REGION Network 171: CIP Return Pump Using P-08.02 (Speed)
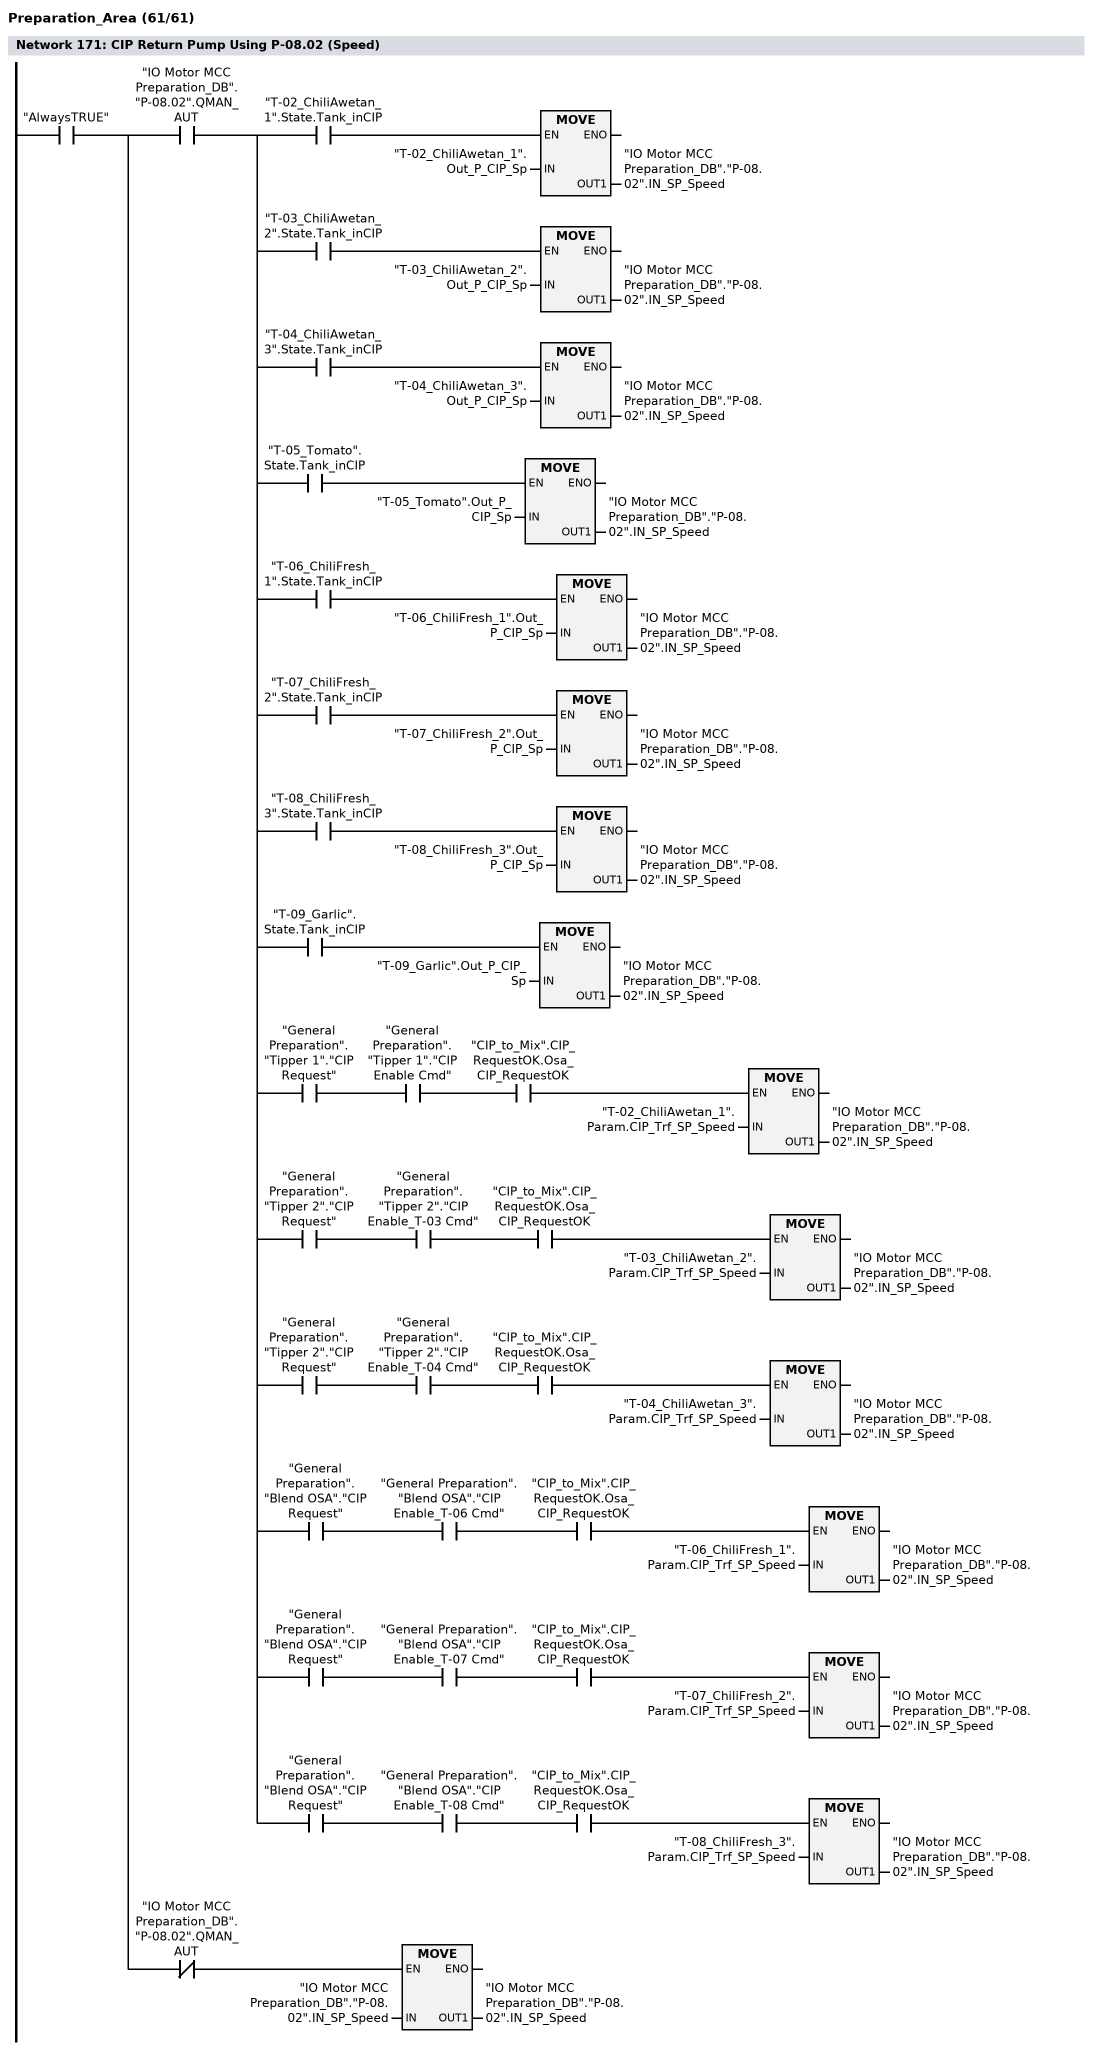
   RUNG wire#powerrail
      Contact( "AlwaysTRUE" )
      wire#w1
      Contact( "IO Motor MCC Preparation_DB"."P-08.02".QMAN_AUT )
      wire#w2
      Contact( "T-02_ChiliAwetan_1".State.Tank_inCIP )
      Move(in := "T-02_ChiliAwetan_1".Out_P_CIP_Sp, out1 => "IO Motor MCC Preparation_DB"."P-08.02".IN_SP_Speed)
   END_RUNG
   RUNG wire#w2
      Contact( "T-03_ChiliAwetan_2".State.Tank_inCIP )
      Move(in := "T-03_ChiliAwetan_2".Out_P_CIP_Sp, out1 => "IO Motor MCC Preparation_DB"."P-08.02".IN_SP_Speed)
   END_RUNG
   RUNG wire#w2
      Contact( "T-04_ChiliAwetan_3".State.Tank_inCIP )
      Move(in := "T-04_ChiliAwetan_3".Out_P_CIP_Sp, out1 => "IO Motor MCC Preparation_DB"."P-08.02".IN_SP_Speed)
   END_RUNG
   RUNG wire#w2
      Contact( "T-05_Tomato".State.Tank_inCIP )
      Move(in := "T-05_Tomato".Out_P_CIP_Sp, out1 => "IO Motor MCC Preparation_DB"."P-08.02".IN_SP_Speed)
   END_RUNG
   RUNG wire#w2
      Contact( "T-06_ChiliFresh_1".State.Tank_inCIP )
      Move(in := "T-06_ChiliFresh_1".Out_P_CIP_Sp, out1 => "IO Motor MCC Preparation_DB"."P-08.02".IN_SP_Speed)
   END_RUNG
   RUNG wire#w2
      Contact( "T-07_ChiliFresh_2".State.Tank_inCIP )
      Move(in := "T-07_ChiliFresh_2".Out_P_CIP_Sp, out1 => "IO Motor MCC Preparation_DB"."P-08.02".IN_SP_Speed)
   END_RUNG
   RUNG wire#w2
      Contact( "T-08_ChiliFresh_3".State.Tank_inCIP )
      Move(in := "T-08_ChiliFresh_3".Out_P_CIP_Sp, out1 => "IO Motor MCC Preparation_DB"."P-08.02".IN_SP_Speed)
   END_RUNG
   RUNG wire#w2
      Contact( "T-09_Garlic".State.Tank_inCIP )
      Move(in := "T-09_Garlic".Out_P_CIP_Sp, out1 => "IO Motor MCC Preparation_DB"."P-08.02".IN_SP_Speed)
   END_RUNG
   RUNG wire#w2
      Contact( "General Preparation"."Tipper 1"."CIP Request" )
      Contact( "General Preparation"."Tipper 1"."CIP Enable Cmd" )
      Contact( "CIP_to_Mix".CIP_RequestOK.Osa_CIP_RequestOK )
      Move(in := "T-02_ChiliAwetan_1".Param.CIP_Trf_SP_Speed, out1 => "IO Motor MCC Preparation_DB"."P-08.02".IN_SP_Speed)
   END_RUNG
   RUNG wire#w2
      Contact( "General Preparation"."Tipper 2"."CIP Request" )
      Contact( "General Preparation"."Tipper 2"."CIP Enable_T-03 Cmd" )
      Contact( "CIP_to_Mix".CIP_RequestOK.Osa_CIP_RequestOK )
      Move(in := "T-03_ChiliAwetan_2".Param.CIP_Trf_SP_Speed, out1 => "IO Motor MCC Preparation_DB"."P-08.02".IN_SP_Speed)
   END_RUNG
   RUNG wire#w2
      Contact( "General Preparation"."Tipper 2"."CIP Request" )
      Contact( "General Preparation"."Tipper 2"."CIP Enable_T-04 Cmd" )
      Contact( "CIP_to_Mix".CIP_RequestOK.Osa_CIP_RequestOK )
      Move(in := "T-04_ChiliAwetan_3".Param.CIP_Trf_SP_Speed, out1 => "IO Motor MCC Preparation_DB"."P-08.02".IN_SP_Speed)
   END_RUNG
   RUNG wire#w2
      Contact( "General Preparation"."Blend OSA"."CIP Request" )
      Contact( "General Preparation"."Blend OSA"."CIP Enable_T-06 Cmd" )
      Contact( "CIP_to_Mix".CIP_RequestOK.Osa_CIP_RequestOK )
      Move(in := "T-06_ChiliFresh_1".Param.CIP_Trf_SP_Speed, out1 => "IO Motor MCC Preparation_DB"."P-08.02".IN_SP_Speed)
   END_RUNG
   RUNG wire#w2
      Contact( "General Preparation"."Blend OSA"."CIP Request" )
      Contact( "General Preparation"."Blend OSA"."CIP Enable_T-07 Cmd" )
      Contact( "CIP_to_Mix".CIP_RequestOK.Osa_CIP_RequestOK )
      Move(in := "T-07_ChiliFresh_2".Param.CIP_Trf_SP_Speed, out1 => "IO Motor MCC Preparation_DB"."P-08.02".IN_SP_Speed)
   END_RUNG
   RUNG wire#w2
      Contact( "General Preparation"."Blend OSA"."CIP Request" )
      Contact( "General Preparation"."Blend OSA"."CIP Enable_T-08 Cmd" )
      Contact( "CIP_to_Mix".CIP_RequestOK.Osa_CIP_RequestOK )
      Move(in := "T-08_ChiliFresh_3".Param.CIP_Trf_SP_Speed, out1 => "IO Motor MCC Preparation_DB"."P-08.02".IN_SP_Speed)
   END_RUNG
   RUNG wire#w1
      I_Contact( "IO Motor MCC Preparation_DB"."P-08.02".QMAN_AUT )
      Move(in := "IO Motor MCC Preparation_DB"."P-08.02".IN_SP_Speed, out1 => "IO Motor MCC Preparation_DB"."P-08.02".IN_SP_Speed)
   END_RUNG
   // the same network as SCL:
   #_w1 := "AlwaysTRUE" AND "IO Motor MCC Preparation_DB"."P-08.02".QMAN_AUT;
   IF #_w1 AND "T-02_ChiliAwetan_1".State.Tank_inCIP THEN
       "IO Motor MCC Preparation_DB"."P-08.02".IN_SP_Speed := "T-02_ChiliAwetan_1".Out_P_CIP_Sp;
   END_IF;
   IF #_w1 AND "T-03_ChiliAwetan_2".State.Tank_inCIP THEN
       "IO Motor MCC Preparation_DB"."P-08.02".IN_SP_Speed := "T-03_ChiliAwetan_2".Out_P_CIP_Sp;
   END_IF;
   IF #_w1 AND "T-04_ChiliAwetan_3".State.Tank_inCIP THEN
       "IO Motor MCC Preparation_DB"."P-08.02".IN_SP_Speed := "T-04_ChiliAwetan_3".Out_P_CIP_Sp;
   END_IF;
   IF #_w1 AND "T-05_Tomato".State.Tank_inCIP THEN
       "IO Motor MCC Preparation_DB"."P-08.02".IN_SP_Speed := "T-05_Tomato".Out_P_CIP_Sp;
   END_IF;
   IF #_w1 AND "T-06_ChiliFresh_1".State.Tank_inCIP THEN
       "IO Motor MCC Preparation_DB"."P-08.02".IN_SP_Speed := "T-06_ChiliFresh_1".Out_P_CIP_Sp;
   END_IF;
   IF #_w1 AND "T-07_ChiliFresh_2".State.Tank_inCIP THEN
       "IO Motor MCC Preparation_DB"."P-08.02".IN_SP_Speed := "T-07_ChiliFresh_2".Out_P_CIP_Sp;
   END_IF;
   IF #_w1 AND "T-08_ChiliFresh_3".State.Tank_inCIP THEN
       "IO Motor MCC Preparation_DB"."P-08.02".IN_SP_Speed := "T-08_ChiliFresh_3".Out_P_CIP_Sp;
   END_IF;
   IF #_w1 AND "T-09_Garlic".State.Tank_inCIP THEN
       "IO Motor MCC Preparation_DB"."P-08.02".IN_SP_Speed := "T-09_Garlic".Out_P_CIP_Sp;
   END_IF;
   IF #_w1 AND "General Preparation"."Tipper 1"."CIP Request" AND "General Preparation"."Tipper 1"."CIP Enable Cmd" AND "CIP_to_Mix".CIP_RequestOK.Osa_CIP_RequestOK THEN
       "IO Motor MCC Preparation_DB"."P-08.02".IN_SP_Speed := "T-02_ChiliAwetan_1".Param.CIP_Trf_SP_Speed;
   END_IF;
   IF #_w1 AND "General Preparation"."Tipper 2"."CIP Request" AND "General Preparation"."Tipper 2"."CIP Enable_T-03 Cmd" AND "CIP_to_Mix".CIP_RequestOK.Osa_CIP_RequestOK THEN
       "IO Motor MCC Preparation_DB"."P-08.02".IN_SP_Speed := "T-03_ChiliAwetan_2".Param.CIP_Trf_SP_Speed;
   END_IF;
   IF #_w1 AND "General Preparation"."Tipper 2"."CIP Request" AND "General Preparation"."Tipper 2"."CIP Enable_T-04 Cmd" AND "CIP_to_Mix".CIP_RequestOK.Osa_CIP_RequestOK THEN
       "IO Motor MCC Preparation_DB"."P-08.02".IN_SP_Speed := "T-04_ChiliAwetan_3".Param.CIP_Trf_SP_Speed;
   END_IF;
   IF #_w1 AND "General Preparation"."Blend OSA"."CIP Request" AND "General Preparation"."Blend OSA"."CIP Enable_T-06 Cmd" AND "CIP_to_Mix".CIP_RequestOK.Osa_CIP_RequestOK THEN
       "IO Motor MCC Preparation_DB"."P-08.02".IN_SP_Speed := "T-06_ChiliFresh_1".Param.CIP_Trf_SP_Speed;
   END_IF;
   IF #_w1 AND "General Preparation"."Blend OSA"."CIP Request" AND "General Preparation"."Blend OSA"."CIP Enable_T-07 Cmd" AND "CIP_to_Mix".CIP_RequestOK.Osa_CIP_RequestOK THEN
       "IO Motor MCC Preparation_DB"."P-08.02".IN_SP_Speed := "T-07_ChiliFresh_2".Param.CIP_Trf_SP_Speed;
   END_IF;
   IF #_w1 AND "General Preparation"."Blend OSA"."CIP Request" AND "General Preparation"."Blend OSA"."CIP Enable_T-08 Cmd" AND "CIP_to_Mix".CIP_RequestOK.Osa_CIP_RequestOK THEN
       "IO Motor MCC Preparation_DB"."P-08.02".IN_SP_Speed := "T-08_ChiliFresh_3".Param.CIP_Trf_SP_Speed;
   END_IF;
   IF "AlwaysTRUE" AND NOT "IO Motor MCC Preparation_DB"."P-08.02".QMAN_AUT THEN
       "IO Motor MCC Preparation_DB"."P-08.02".IN_SP_Speed := "IO Motor MCC Preparation_DB"."P-08.02".IN_SP_Speed;
   END_IF;
END_REGION

NETWORK
TITLE = Valve IO
//Valve T-02.01 Chili Awetan Tank 1
      CALL  "IO Valve T02 Chili", "IO_Valve_T02_Chili"
      ( lock    := ,
        Init    := "General_DB".Initial,
        testing := "General_DB"."Testing FB Valve".Preparation,
        Reset   := "General_DB".Reset
      );
//Valve T-03.01 Chili Awetan Tank 2
      CALL  "IO Valve T03 Chili", "IO_Valve_T03_Chili"
      ( lock    := ,
        Init    := "General_DB".Initial,
        testing := "General_DB"."Testing FB Valve".Preparation,
        Reset   := "General_DB".Reset
      );
//Valve T-04.01 Chili Awetan Tank 3
      CALL  "IO Valve T04 Chili", "IO_Valve_T04_Chili"
      ( lock    := ,
        Init    := "General_DB".Initial,
        testing := "General_DB"."Testing FB Valve".Preparation,
        Reset   := "General_DB".Reset
      );
//Valve T-05.01 Tomato Tank
      CALL  "IO Valve T05 Tomato", "IO_Valve_T05_Tomato"
      ( lock    := ,
        Init    := "General_DB".Initial,
        testing := "General_DB"."Testing FB Valve".Preparation,
        Reset   := "General_DB".Reset
      );
//Valve T-06.01 Fresh Chili Tank 1
      CALL  "IO Valve T06 FreshChili", "IO_Valve_T06_FreshChili"
      ( lock    := ,
        Init    := "General_DB".Initial,
        testing := "General_DB"."Testing FB Valve".Preparation,
        Reset   := "General_DB".Reset
      );
//Valve T-07.01 Fresh Chili Tank 2
      CALL  "IO Valve T07 FreshChili", "IO_Valve_T07_FreshChili"
      ( lock    := ,
        Init    := "General_DB".Initial,
        testing := "General_DB"."Testing FB Valve".Preparation,
        Reset   := "General_DB".Reset
      );
//Valve T-08.01 Fresh Chili Tank 3
      CALL  "IO Valve T08 FreshChili", "IO_Valve_T08_FreshChili"
      ( lock    := ,
        Init    := "General_DB".Initial,
        testing := "General_DB"."Testing FB Valve".Preparation,
        Reset   := "General_DB".Reset
      );
//Valve T-09.01 Garlic Tank
      CALL  "IO Valve T09 Garlic", "IO_Valve_T09_Garlic"
      ( lock    := ,
        Init    := "General_DB".Initial,
        testing := "General_DB"."Testing FB Valve".Preparation,
        Reset   := "General_DB".Reset
      );
//Valve T-10.01 Vinegar Tank
      CALL  "IO Valve T10 Vinegar", "IO_Valve_T10_Vinegar"
      ( lock    := ,
        Init    := "General_DB".Initial,
        testing := "General_DB"."Testing FB Valve".Preparation,
        Reset   := "General_DB".Reset
      );
//Valve T-10.01 HotWater
      CALL  "IO Valve T51 HotWaterLine", "IO_Valve_T51_HW"
      ( lock    := ,
        Init    := "General_DB".Initial,
        testing := "General_DB"."Testing FB Valve".Preparation,
        Reset   := "General_DB".Reset
      );


END_FUNCTION

FUNCTION_BLOCK "IO Analog Preparation"   // FB12, LAD
{ S7_Optimized_Access := 'FALSE' }
VERSION : 0.1
// stored: AutoNumber true, IsIECCheckEnabled false, SetENOAutomatically false, UDAEnableTagReadback false
   VAR_INPUT
      Init : Bool;
      Reset : Bool;
   END_VAR
   VAR
      "LT-01.01" : "Ana_w_K1K2";   // LEVEL TRANSMITTER HOT WATER TANK T-01.00
      "TT-01.01" : "Ana_w_K1K2";   // TEMP. TRANSMITTER HOT WATER TANK T-01.00
      "TT-01.02" : "Ana_w_K1K2";   // TEMP.TRANSMITTER LINE HOT WATER
      "LT-02.01" : "Ana_w_K1K2";   // LEVEL TRANSMITTER BUFFER TANK CHILI AWETAN T-02.00
      "LT-03.01" : "Ana_w_K1K2";   // LEVEL TRANSMITTER BUFFER TANK CHILI AWETAN T-03.00
      "LT-04.01" : "Ana_w_K1K2";   // LEVEL TRANSMITTER BUFFER TANK CHILI AWETAN T-04.00
      "LT-05.01" : "Ana_w_K1K2";   // LEVEL TRANSMITTER BUFFER TANK TOMATO T-05.00
      "LT-06.01" : "Ana_w_K1K2";   // LEVEL TRANSMITTER BUFFER TANK CHILI FRESH T-06.00
      "LT-07.01" : "Ana_w_K1K2";   // LEVEL TRANSMITTER BUFFER TANK CHILI FRESH T-07.00
      "LT-08.01" : "Ana_w_K1K2";   // LEVEL TRANSMITTER BUFFER TANK CHILI FRESH T-08.00
      "LT-09.01" : "Ana_w_K1K2";   // LEVEL TRANSMITTER BUFFER TANK GARLIC T-09.00
      "LT-10.01" : "Ana_w_K1K2";   // LEVEL TRANSMITTER BUFFER TANK GARLIC T-10.00
      "TT-51.01" { S7_SetPoint := 'True'} : "Ana_w_K1K2";
      "CV-51.11" { S7_SetPoint := 'True'} : "Ana_w_K1K2";
      "FT-51.01" { S7_SetPoint := 'True'} : "Ana_w_K1K2";
      "FT-02.01" { S7_SetPoint := 'True'} : "Ana_w_K1K2";
      "FT-02.01Com" { S7_SetPoint := 'True'} : "Read FT Comm";
      "FT-03.01" { S7_SetPoint := 'True'} : "Ana_w_K1K2";
      "FT-03.01Com" { S7_SetPoint := 'True'} : "Read FT Comm";
      "FT-04.01" { S7_SetPoint := 'True'} : "Ana_w_K1K2";
      "FT-04.01Com" { S7_SetPoint := 'True'} : "Read FT Comm";
      "FT-05.01" { S7_SetPoint := 'True'} : "Ana_w_K1K2";
      "FT-05.01Com" { S7_SetPoint := 'True'} : "Read FT Comm";
      "FT-06.01" { S7_SetPoint := 'True'} : "Ana_w_K1K2";
      "FT-06.01Com" { S7_SetPoint := 'True'} : "Read FT Comm";
      "FT-07.01" { S7_SetPoint := 'True'} : "Ana_w_K1K2";
      "FT-07.01Com" { S7_SetPoint := 'True'} : "Read FT Comm";
      "FT-08.01" { S7_SetPoint := 'True'} : "Ana_w_K1K2";
      "FT-08.01Com" { S7_SetPoint := 'True'} : "Read FT Comm";
      "FT-09.01" { S7_SetPoint := 'True'} : "Ana_w_K1K2";
      "FT-09.01Com" { S7_SetPoint := 'True'} : "Read FT Comm";
      "FT-10.01" { S7_SetPoint := 'True'} : "Ana_w_K1K2";
      "FT-10.01Com" { S7_SetPoint := 'True'} : "Read FT Comm";
   END_VAR
BEGIN

REGION Network 1: LT-01.01
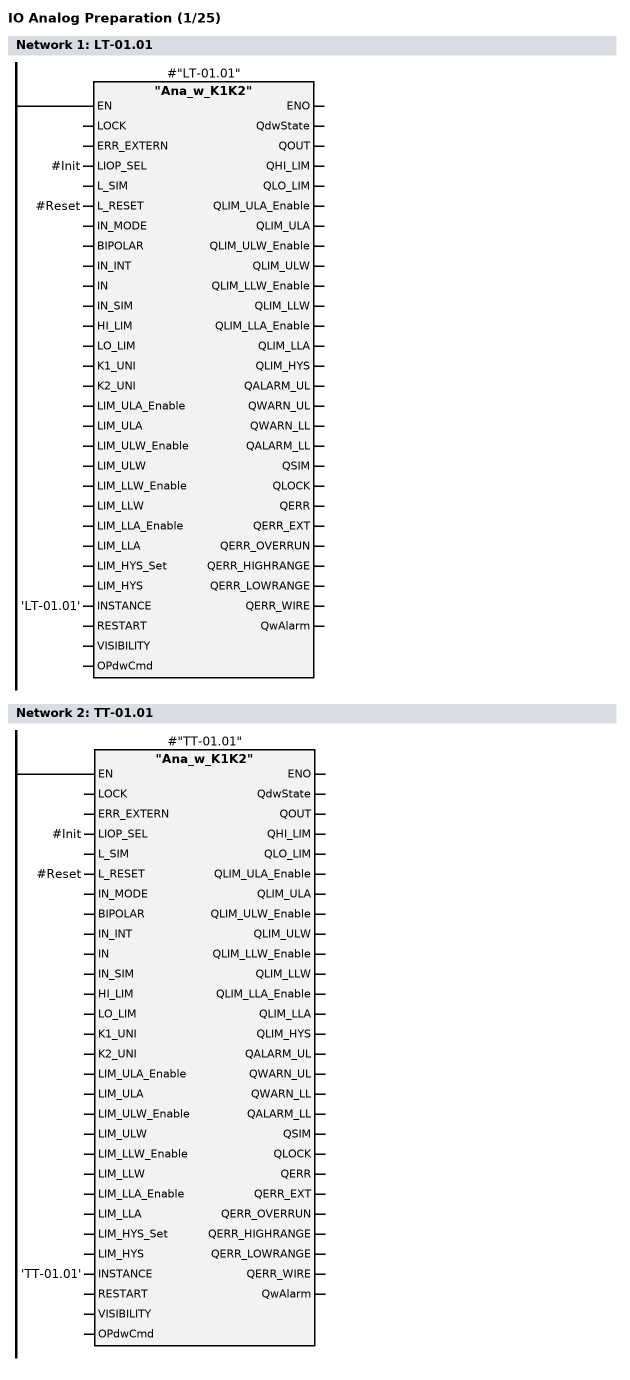
   RUNG wire#powerrail
      #"LT-01.01"(LOCK :=, ERR_EXTERN :=, LIOP_SEL := #Init, L_SIM :=, L_RESET := #Reset, IN_MODE :=, BIPOLAR :=, IN_INT :=, IN :=, IN_SIM :=, HI_LIM :=, LO_LIM :=, K1_UNI :=, K2_UNI :=, LIM_ULA_Enable :=, LIM_ULA :=, LIM_ULW_Enable :=, LIM_ULW :=, LIM_LLW_Enable :=, LIM_LLW :=, LIM_LLA_Enable :=, LIM_LLA :=, LIM_HYS_Set :=, LIM_HYS :=, INSTANCE := 'LT-01.01', RESTART :=, VISIBILITY :=, OPdwCmd :=, QdwState =>, QOUT =>, QHI_LIM =>, QLO_LIM =>, QLIM_ULA_Enable =>, QLIM_ULA =>, QLIM_ULW_Enable =>, QLIM_ULW =>, QLIM_LLW_Enable =>, QLIM_LLW =>, QLIM_LLA_Enable =>, QLIM_LLA =>, QLIM_HYS =>, QALARM_UL =>, QWARN_UL =>, QWARN_LL =>, QALARM_LL =>, QSIM =>, QLOCK =>, QERR =>, QERR_EXT =>, QERR_OVERRUN =>, QERR_HIGHRANGE =>, QERR_LOWRANGE =>, QERR_WIRE =>, QwAlarm =>)
   END_RUNG
   // the same network as SCL:
   #"LT-01.01"(LIOP_SEL := #Init, L_RESET := #Reset, INSTANCE := 'LT-01.01');   // "Ana_w_K1K2"
END_REGION

REGION Network 2: TT-01.01
   RUNG wire#powerrail
      #"TT-01.01"(LOCK :=, ERR_EXTERN :=, LIOP_SEL := #Init, L_SIM :=, L_RESET := #Reset, IN_MODE :=, BIPOLAR :=, IN_INT :=, IN :=, IN_SIM :=, HI_LIM :=, LO_LIM :=, K1_UNI :=, K2_UNI :=, LIM_ULA_Enable :=, LIM_ULA :=, LIM_ULW_Enable :=, LIM_ULW :=, LIM_LLW_Enable :=, LIM_LLW :=, LIM_LLA_Enable :=, LIM_LLA :=, LIM_HYS_Set :=, LIM_HYS :=, INSTANCE := 'TT-01.01', RESTART :=, VISIBILITY :=, OPdwCmd :=, QdwState =>, QOUT =>, QHI_LIM =>, QLO_LIM =>, QLIM_ULA_Enable =>, QLIM_ULA =>, QLIM_ULW_Enable =>, QLIM_ULW =>, QLIM_LLW_Enable =>, QLIM_LLW =>, QLIM_LLA_Enable =>, QLIM_LLA =>, QLIM_HYS =>, QALARM_UL =>, QWARN_UL =>, QWARN_LL =>, QALARM_LL =>, QSIM =>, QLOCK =>, QERR =>, QERR_EXT =>, QERR_OVERRUN =>, QERR_HIGHRANGE =>, QERR_LOWRANGE =>, QERR_WIRE =>, QwAlarm =>)
   END_RUNG
   // the same network as SCL:
   #"TT-01.01"(LIOP_SEL := #Init, L_RESET := #Reset, INSTANCE := 'TT-01.01');   // "Ana_w_K1K2"
END_REGION

REGION Network 3: TT-01.02
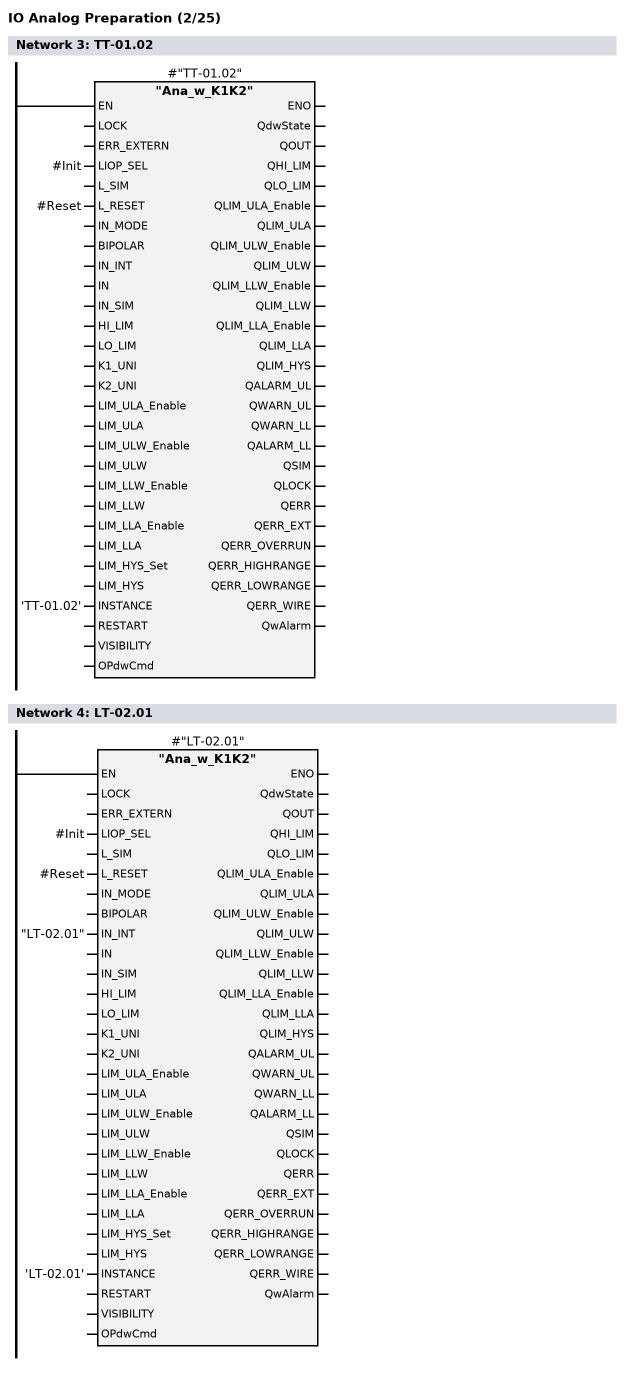
   RUNG wire#powerrail
      #"TT-01.02"(LOCK :=, ERR_EXTERN :=, LIOP_SEL := #Init, L_SIM :=, L_RESET := #Reset, IN_MODE :=, BIPOLAR :=, IN_INT :=, IN :=, IN_SIM :=, HI_LIM :=, LO_LIM :=, K1_UNI :=, K2_UNI :=, LIM_ULA_Enable :=, LIM_ULA :=, LIM_ULW_Enable :=, LIM_ULW :=, LIM_LLW_Enable :=, LIM_LLW :=, LIM_LLA_Enable :=, LIM_LLA :=, LIM_HYS_Set :=, LIM_HYS :=, INSTANCE := 'TT-01.02', RESTART :=, VISIBILITY :=, OPdwCmd :=, QdwState =>, QOUT =>, QHI_LIM =>, QLO_LIM =>, QLIM_ULA_Enable =>, QLIM_ULA =>, QLIM_ULW_Enable =>, QLIM_ULW =>, QLIM_LLW_Enable =>, QLIM_LLW =>, QLIM_LLA_Enable =>, QLIM_LLA =>, QLIM_HYS =>, QALARM_UL =>, QWARN_UL =>, QWARN_LL =>, QALARM_LL =>, QSIM =>, QLOCK =>, QERR =>, QERR_EXT =>, QERR_OVERRUN =>, QERR_HIGHRANGE =>, QERR_LOWRANGE =>, QERR_WIRE =>, QwAlarm =>)
   END_RUNG
   // the same network as SCL:
   #"TT-01.02"(LIOP_SEL := #Init, L_RESET := #Reset, INSTANCE := 'TT-01.02');   // "Ana_w_K1K2"
END_REGION

REGION Network 4: LT-02.01
   RUNG wire#powerrail
      #"LT-02.01"(LOCK :=, ERR_EXTERN :=, LIOP_SEL := #Init, L_SIM :=, L_RESET := #Reset, IN_MODE :=, BIPOLAR :=, IN_INT := "LT-02.01", IN :=, IN_SIM :=, HI_LIM :=, LO_LIM :=, K1_UNI :=, K2_UNI :=, LIM_ULA_Enable :=, LIM_ULA :=, LIM_ULW_Enable :=, LIM_ULW :=, LIM_LLW_Enable :=, LIM_LLW :=, LIM_LLA_Enable :=, LIM_LLA :=, LIM_HYS_Set :=, LIM_HYS :=, INSTANCE := 'LT-02.01', RESTART :=, VISIBILITY :=, OPdwCmd :=, QdwState =>, QOUT =>, QHI_LIM =>, QLO_LIM =>, QLIM_ULA_Enable =>, QLIM_ULA =>, QLIM_ULW_Enable =>, QLIM_ULW =>, QLIM_LLW_Enable =>, QLIM_LLW =>, QLIM_LLA_Enable =>, QLIM_LLA =>, QLIM_HYS =>, QALARM_UL =>, QWARN_UL =>, QWARN_LL =>, QALARM_LL =>, QSIM =>, QLOCK =>, QERR =>, QERR_EXT =>, QERR_OVERRUN =>, QERR_HIGHRANGE =>, QERR_LOWRANGE =>, QERR_WIRE =>, QwAlarm =>)
   END_RUNG
   // the same network as SCL:
   #"LT-02.01"(LIOP_SEL := #Init, L_RESET := #Reset, IN_INT := "LT-02.01", INSTANCE := 'LT-02.01');   // "Ana_w_K1K2"
END_REGION

REGION Network 5: LT-03.01
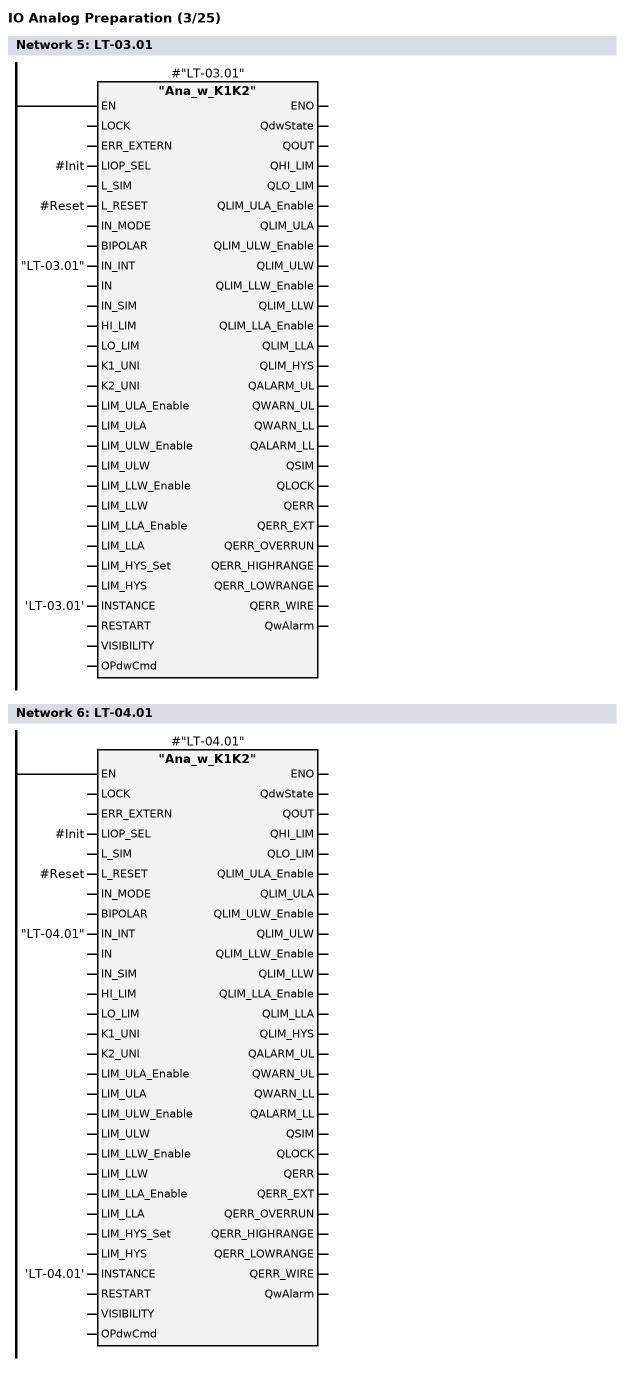
   RUNG wire#powerrail
      #"LT-03.01"(LOCK :=, ERR_EXTERN :=, LIOP_SEL := #Init, L_SIM :=, L_RESET := #Reset, IN_MODE :=, BIPOLAR :=, IN_INT := "LT-03.01", IN :=, IN_SIM :=, HI_LIM :=, LO_LIM :=, K1_UNI :=, K2_UNI :=, LIM_ULA_Enable :=, LIM_ULA :=, LIM_ULW_Enable :=, LIM_ULW :=, LIM_LLW_Enable :=, LIM_LLW :=, LIM_LLA_Enable :=, LIM_LLA :=, LIM_HYS_Set :=, LIM_HYS :=, INSTANCE := 'LT-03.01', RESTART :=, VISIBILITY :=, OPdwCmd :=, QdwState =>, QOUT =>, QHI_LIM =>, QLO_LIM =>, QLIM_ULA_Enable =>, QLIM_ULA =>, QLIM_ULW_Enable =>, QLIM_ULW =>, QLIM_LLW_Enable =>, QLIM_LLW =>, QLIM_LLA_Enable =>, QLIM_LLA =>, QLIM_HYS =>, QALARM_UL =>, QWARN_UL =>, QWARN_LL =>, QALARM_LL =>, QSIM =>, QLOCK =>, QERR =>, QERR_EXT =>, QERR_OVERRUN =>, QERR_HIGHRANGE =>, QERR_LOWRANGE =>, QERR_WIRE =>, QwAlarm =>)
   END_RUNG
   // the same network as SCL:
   #"LT-03.01"(LIOP_SEL := #Init, L_RESET := #Reset, IN_INT := "LT-03.01", INSTANCE := 'LT-03.01');   // "Ana_w_K1K2"
END_REGION

REGION Network 6: LT-04.01
   RUNG wire#powerrail
      #"LT-04.01"(LOCK :=, ERR_EXTERN :=, LIOP_SEL := #Init, L_SIM :=, L_RESET := #Reset, IN_MODE :=, BIPOLAR :=, IN_INT := "LT-04.01", IN :=, IN_SIM :=, HI_LIM :=, LO_LIM :=, K1_UNI :=, K2_UNI :=, LIM_ULA_Enable :=, LIM_ULA :=, LIM_ULW_Enable :=, LIM_ULW :=, LIM_LLW_Enable :=, LIM_LLW :=, LIM_LLA_Enable :=, LIM_LLA :=, LIM_HYS_Set :=, LIM_HYS :=, INSTANCE := 'LT-04.01', RESTART :=, VISIBILITY :=, OPdwCmd :=, QdwState =>, QOUT =>, QHI_LIM =>, QLO_LIM =>, QLIM_ULA_Enable =>, QLIM_ULA =>, QLIM_ULW_Enable =>, QLIM_ULW =>, QLIM_LLW_Enable =>, QLIM_LLW =>, QLIM_LLA_Enable =>, QLIM_LLA =>, QLIM_HYS =>, QALARM_UL =>, QWARN_UL =>, QWARN_LL =>, QALARM_LL =>, QSIM =>, QLOCK =>, QERR =>, QERR_EXT =>, QERR_OVERRUN =>, QERR_HIGHRANGE =>, QERR_LOWRANGE =>, QERR_WIRE =>, QwAlarm =>)
   END_RUNG
   // the same network as SCL:
   #"LT-04.01"(LIOP_SEL := #Init, L_RESET := #Reset, IN_INT := "LT-04.01", INSTANCE := 'LT-04.01');   // "Ana_w_K1K2"
END_REGION

REGION Network 7: LT-05.01
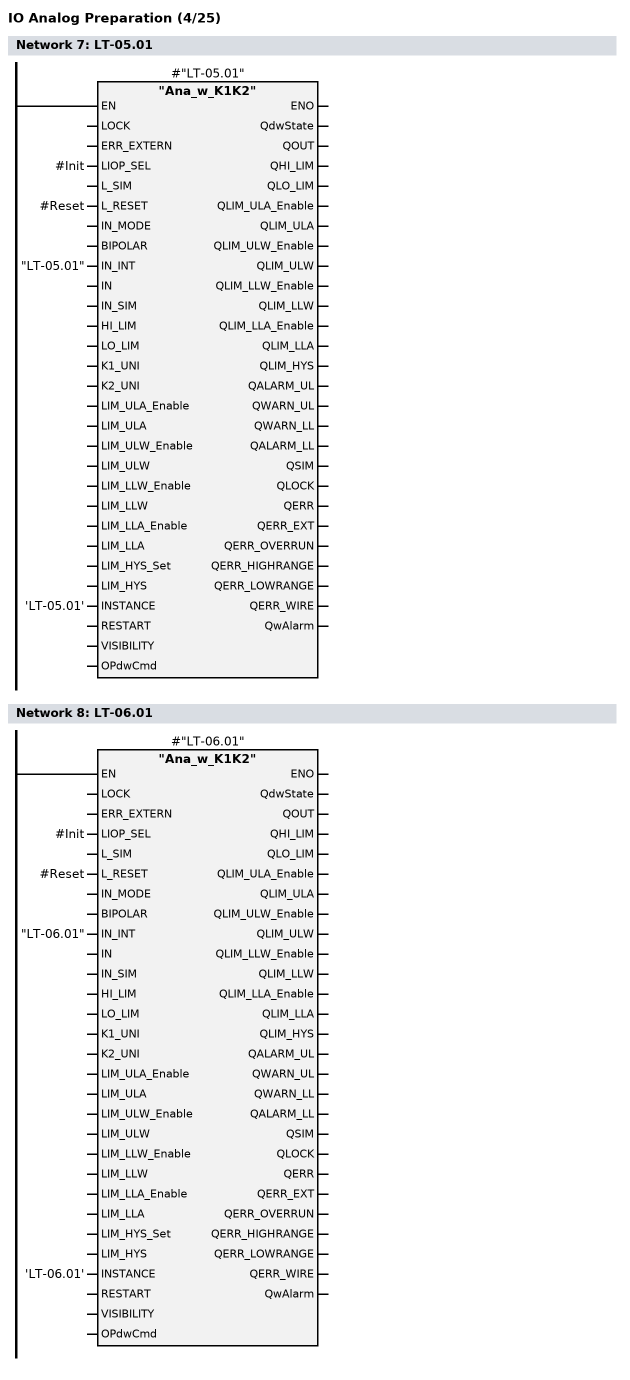
   RUNG wire#powerrail
      #"LT-05.01"(LOCK :=, ERR_EXTERN :=, LIOP_SEL := #Init, L_SIM :=, L_RESET := #Reset, IN_MODE :=, BIPOLAR :=, IN_INT := "LT-05.01", IN :=, IN_SIM :=, HI_LIM :=, LO_LIM :=, K1_UNI :=, K2_UNI :=, LIM_ULA_Enable :=, LIM_ULA :=, LIM_ULW_Enable :=, LIM_ULW :=, LIM_LLW_Enable :=, LIM_LLW :=, LIM_LLA_Enable :=, LIM_LLA :=, LIM_HYS_Set :=, LIM_HYS :=, INSTANCE := 'LT-05.01', RESTART :=, VISIBILITY :=, OPdwCmd :=, QdwState =>, QOUT =>, QHI_LIM =>, QLO_LIM =>, QLIM_ULA_Enable =>, QLIM_ULA =>, QLIM_ULW_Enable =>, QLIM_ULW =>, QLIM_LLW_Enable =>, QLIM_LLW =>, QLIM_LLA_Enable =>, QLIM_LLA =>, QLIM_HYS =>, QALARM_UL =>, QWARN_UL =>, QWARN_LL =>, QALARM_LL =>, QSIM =>, QLOCK =>, QERR =>, QERR_EXT =>, QERR_OVERRUN =>, QERR_HIGHRANGE =>, QERR_LOWRANGE =>, QERR_WIRE =>, QwAlarm =>)
   END_RUNG
   // the same network as SCL:
   #"LT-05.01"(LIOP_SEL := #Init, L_RESET := #Reset, IN_INT := "LT-05.01", INSTANCE := 'LT-05.01');   // "Ana_w_K1K2"
END_REGION

REGION Network 8: LT-06.01
   RUNG wire#powerrail
      #"LT-06.01"(LOCK :=, ERR_EXTERN :=, LIOP_SEL := #Init, L_SIM :=, L_RESET := #Reset, IN_MODE :=, BIPOLAR :=, IN_INT := "LT-06.01", IN :=, IN_SIM :=, HI_LIM :=, LO_LIM :=, K1_UNI :=, K2_UNI :=, LIM_ULA_Enable :=, LIM_ULA :=, LIM_ULW_Enable :=, LIM_ULW :=, LIM_LLW_Enable :=, LIM_LLW :=, LIM_LLA_Enable :=, LIM_LLA :=, LIM_HYS_Set :=, LIM_HYS :=, INSTANCE := 'LT-06.01', RESTART :=, VISIBILITY :=, OPdwCmd :=, QdwState =>, QOUT =>, QHI_LIM =>, QLO_LIM =>, QLIM_ULA_Enable =>, QLIM_ULA =>, QLIM_ULW_Enable =>, QLIM_ULW =>, QLIM_LLW_Enable =>, QLIM_LLW =>, QLIM_LLA_Enable =>, QLIM_LLA =>, QLIM_HYS =>, QALARM_UL =>, QWARN_UL =>, QWARN_LL =>, QALARM_LL =>, QSIM =>, QLOCK =>, QERR =>, QERR_EXT =>, QERR_OVERRUN =>, QERR_HIGHRANGE =>, QERR_LOWRANGE =>, QERR_WIRE =>, QwAlarm =>)
   END_RUNG
   // the same network as SCL:
   #"LT-06.01"(LIOP_SEL := #Init, L_RESET := #Reset, IN_INT := "LT-06.01", INSTANCE := 'LT-06.01');   // "Ana_w_K1K2"
END_REGION

REGION Network 9: LT-07.01
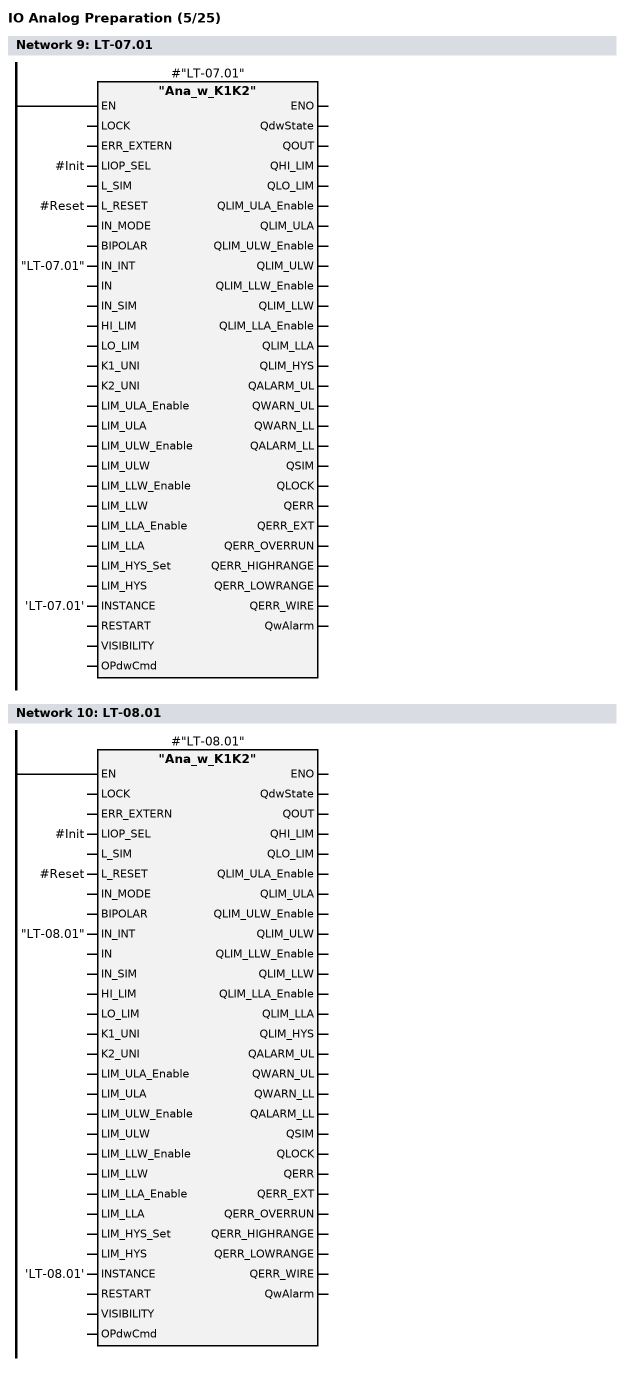
   RUNG wire#powerrail
      #"LT-07.01"(LOCK :=, ERR_EXTERN :=, LIOP_SEL := #Init, L_SIM :=, L_RESET := #Reset, IN_MODE :=, BIPOLAR :=, IN_INT := "LT-07.01", IN :=, IN_SIM :=, HI_LIM :=, LO_LIM :=, K1_UNI :=, K2_UNI :=, LIM_ULA_Enable :=, LIM_ULA :=, LIM_ULW_Enable :=, LIM_ULW :=, LIM_LLW_Enable :=, LIM_LLW :=, LIM_LLA_Enable :=, LIM_LLA :=, LIM_HYS_Set :=, LIM_HYS :=, INSTANCE := 'LT-07.01', RESTART :=, VISIBILITY :=, OPdwCmd :=, QdwState =>, QOUT =>, QHI_LIM =>, QLO_LIM =>, QLIM_ULA_Enable =>, QLIM_ULA =>, QLIM_ULW_Enable =>, QLIM_ULW =>, QLIM_LLW_Enable =>, QLIM_LLW =>, QLIM_LLA_Enable =>, QLIM_LLA =>, QLIM_HYS =>, QALARM_UL =>, QWARN_UL =>, QWARN_LL =>, QALARM_LL =>, QSIM =>, QLOCK =>, QERR =>, QERR_EXT =>, QERR_OVERRUN =>, QERR_HIGHRANGE =>, QERR_LOWRANGE =>, QERR_WIRE =>, QwAlarm =>)
   END_RUNG
   // the same network as SCL:
   #"LT-07.01"(LIOP_SEL := #Init, L_RESET := #Reset, IN_INT := "LT-07.01", INSTANCE := 'LT-07.01');   // "Ana_w_K1K2"
END_REGION

REGION Network 10: LT-08.01
   RUNG wire#powerrail
      #"LT-08.01"(LOCK :=, ERR_EXTERN :=, LIOP_SEL := #Init, L_SIM :=, L_RESET := #Reset, IN_MODE :=, BIPOLAR :=, IN_INT := "LT-08.01", IN :=, IN_SIM :=, HI_LIM :=, LO_LIM :=, K1_UNI :=, K2_UNI :=, LIM_ULA_Enable :=, LIM_ULA :=, LIM_ULW_Enable :=, LIM_ULW :=, LIM_LLW_Enable :=, LIM_LLW :=, LIM_LLA_Enable :=, LIM_LLA :=, LIM_HYS_Set :=, LIM_HYS :=, INSTANCE := 'LT-08.01', RESTART :=, VISIBILITY :=, OPdwCmd :=, QdwState =>, QOUT =>, QHI_LIM =>, QLO_LIM =>, QLIM_ULA_Enable =>, QLIM_ULA =>, QLIM_ULW_Enable =>, QLIM_ULW =>, QLIM_LLW_Enable =>, QLIM_LLW =>, QLIM_LLA_Enable =>, QLIM_LLA =>, QLIM_HYS =>, QALARM_UL =>, QWARN_UL =>, QWARN_LL =>, QALARM_LL =>, QSIM =>, QLOCK =>, QERR =>, QERR_EXT =>, QERR_OVERRUN =>, QERR_HIGHRANGE =>, QERR_LOWRANGE =>, QERR_WIRE =>, QwAlarm =>)
   END_RUNG
   // the same network as SCL:
   #"LT-08.01"(LIOP_SEL := #Init, L_RESET := #Reset, IN_INT := "LT-08.01", INSTANCE := 'LT-08.01');   // "Ana_w_K1K2"
END_REGION

REGION Network 11: LT-09.01
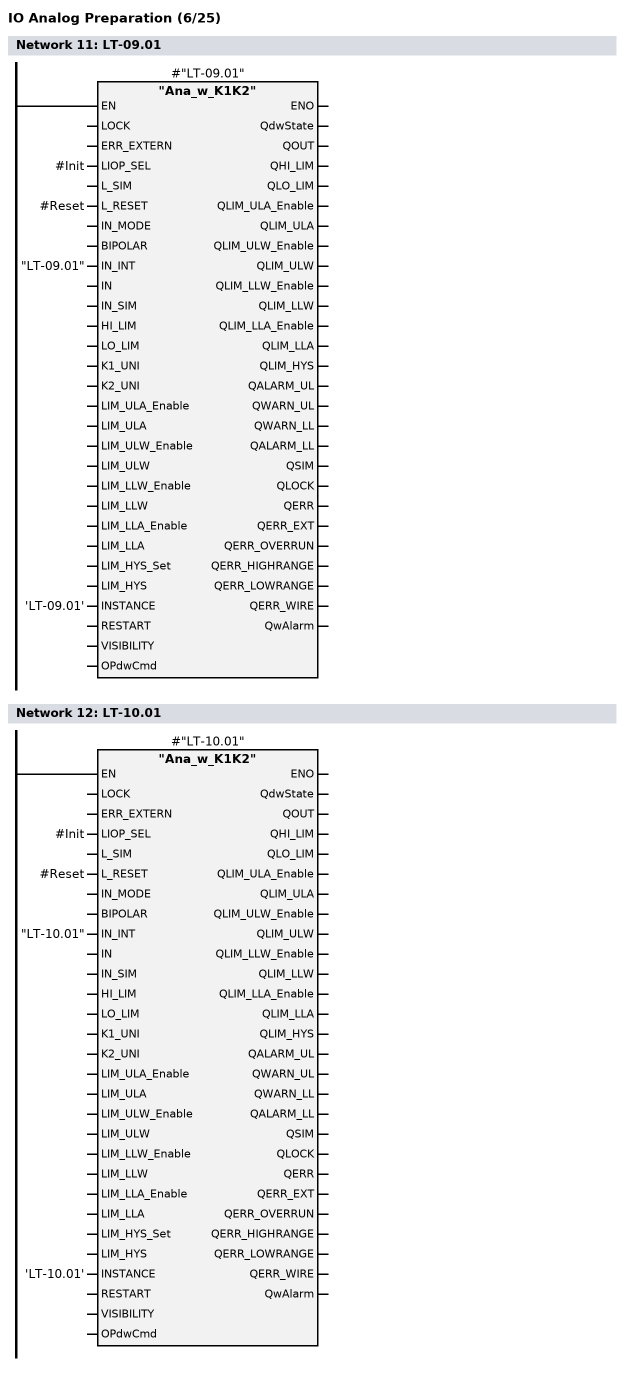
   RUNG wire#powerrail
      #"LT-09.01"(LOCK :=, ERR_EXTERN :=, LIOP_SEL := #Init, L_SIM :=, L_RESET := #Reset, IN_MODE :=, BIPOLAR :=, IN_INT := "LT-09.01", IN :=, IN_SIM :=, HI_LIM :=, LO_LIM :=, K1_UNI :=, K2_UNI :=, LIM_ULA_Enable :=, LIM_ULA :=, LIM_ULW_Enable :=, LIM_ULW :=, LIM_LLW_Enable :=, LIM_LLW :=, LIM_LLA_Enable :=, LIM_LLA :=, LIM_HYS_Set :=, LIM_HYS :=, INSTANCE := 'LT-09.01', RESTART :=, VISIBILITY :=, OPdwCmd :=, QdwState =>, QOUT =>, QHI_LIM =>, QLO_LIM =>, QLIM_ULA_Enable =>, QLIM_ULA =>, QLIM_ULW_Enable =>, QLIM_ULW =>, QLIM_LLW_Enable =>, QLIM_LLW =>, QLIM_LLA_Enable =>, QLIM_LLA =>, QLIM_HYS =>, QALARM_UL =>, QWARN_UL =>, QWARN_LL =>, QALARM_LL =>, QSIM =>, QLOCK =>, QERR =>, QERR_EXT =>, QERR_OVERRUN =>, QERR_HIGHRANGE =>, QERR_LOWRANGE =>, QERR_WIRE =>, QwAlarm =>)
   END_RUNG
   // the same network as SCL:
   #"LT-09.01"(LIOP_SEL := #Init, L_RESET := #Reset, IN_INT := "LT-09.01", INSTANCE := 'LT-09.01');   // "Ana_w_K1K2"
END_REGION

REGION Network 12: LT-10.01
   RUNG wire#powerrail
      #"LT-10.01"(LOCK :=, ERR_EXTERN :=, LIOP_SEL := #Init, L_SIM :=, L_RESET := #Reset, IN_MODE :=, BIPOLAR :=, IN_INT := "LT-10.01", IN :=, IN_SIM :=, HI_LIM :=, LO_LIM :=, K1_UNI :=, K2_UNI :=, LIM_ULA_Enable :=, LIM_ULA :=, LIM_ULW_Enable :=, LIM_ULW :=, LIM_LLW_Enable :=, LIM_LLW :=, LIM_LLA_Enable :=, LIM_LLA :=, LIM_HYS_Set :=, LIM_HYS :=, INSTANCE := 'LT-10.01', RESTART :=, VISIBILITY :=, OPdwCmd :=, QdwState =>, QOUT =>, QHI_LIM =>, QLO_LIM =>, QLIM_ULA_Enable =>, QLIM_ULA =>, QLIM_ULW_Enable =>, QLIM_ULW =>, QLIM_LLW_Enable =>, QLIM_LLW =>, QLIM_LLA_Enable =>, QLIM_LLA =>, QLIM_HYS =>, QALARM_UL =>, QWARN_UL =>, QWARN_LL =>, QALARM_LL =>, QSIM =>, QLOCK =>, QERR =>, QERR_EXT =>, QERR_OVERRUN =>, QERR_HIGHRANGE =>, QERR_LOWRANGE =>, QERR_WIRE =>, QwAlarm =>)
   END_RUNG
   // the same network as SCL:
   #"LT-10.01"(LIOP_SEL := #Init, L_RESET := #Reset, IN_INT := "LT-10.01", INSTANCE := 'LT-10.01');   // "Ana_w_K1K2"
END_REGION

REGION Network 13: TT-51.01
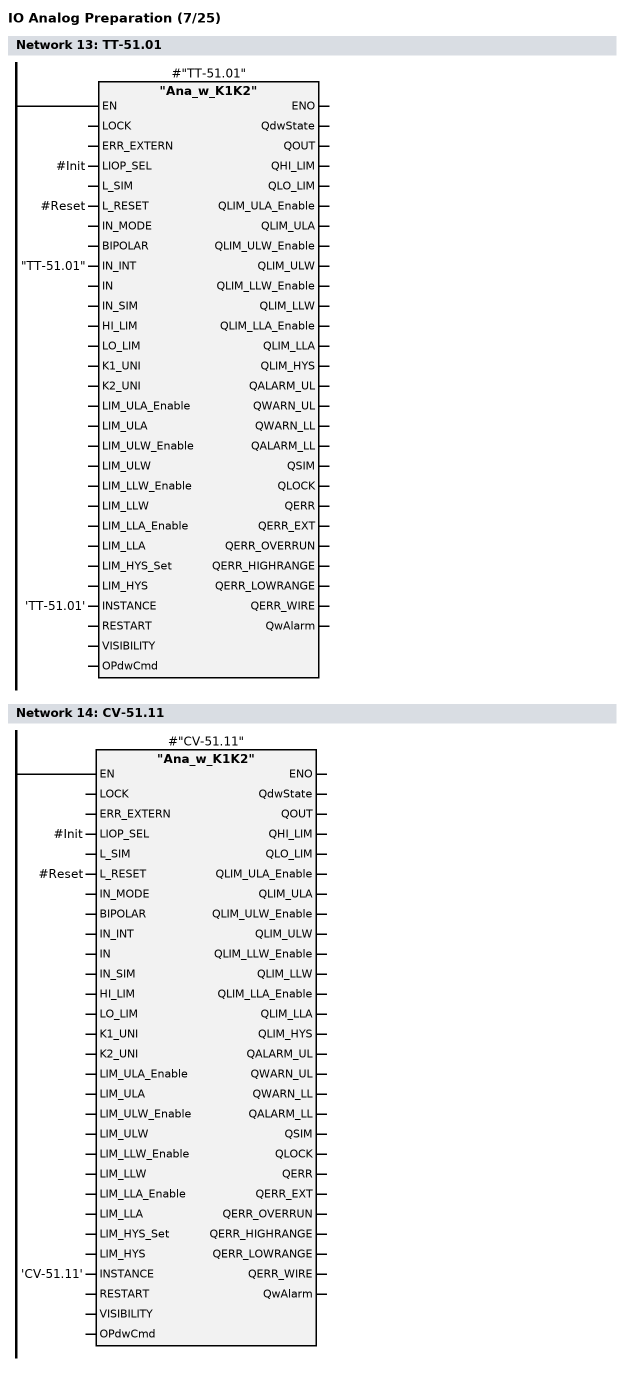
   RUNG wire#powerrail
      #"TT-51.01"(LOCK :=, ERR_EXTERN :=, LIOP_SEL := #Init, L_SIM :=, L_RESET := #Reset, IN_MODE :=, BIPOLAR :=, IN_INT := "TT-51.01", IN :=, IN_SIM :=, HI_LIM :=, LO_LIM :=, K1_UNI :=, K2_UNI :=, LIM_ULA_Enable :=, LIM_ULA :=, LIM_ULW_Enable :=, LIM_ULW :=, LIM_LLW_Enable :=, LIM_LLW :=, LIM_LLA_Enable :=, LIM_LLA :=, LIM_HYS_Set :=, LIM_HYS :=, INSTANCE := 'TT-51.01', RESTART :=, VISIBILITY :=, OPdwCmd :=, QdwState =>, QOUT =>, QHI_LIM =>, QLO_LIM =>, QLIM_ULA_Enable =>, QLIM_ULA =>, QLIM_ULW_Enable =>, QLIM_ULW =>, QLIM_LLW_Enable =>, QLIM_LLW =>, QLIM_LLA_Enable =>, QLIM_LLA =>, QLIM_HYS =>, QALARM_UL =>, QWARN_UL =>, QWARN_LL =>, QALARM_LL =>, QSIM =>, QLOCK =>, QERR =>, QERR_EXT =>, QERR_OVERRUN =>, QERR_HIGHRANGE =>, QERR_LOWRANGE =>, QERR_WIRE =>, QwAlarm =>)
   END_RUNG
   // the same network as SCL:
   #"TT-51.01"(LIOP_SEL := #Init, L_RESET := #Reset, IN_INT := "TT-51.01", INSTANCE := 'TT-51.01');   // "Ana_w_K1K2"
END_REGION

REGION Network 14: CV-51.11
   RUNG wire#powerrail
      #"CV-51.11"(LOCK :=, ERR_EXTERN :=, LIOP_SEL := #Init, L_SIM :=, L_RESET := #Reset, IN_MODE :=, BIPOLAR :=, IN_INT :=, IN :=, IN_SIM :=, HI_LIM :=, LO_LIM :=, K1_UNI :=, K2_UNI :=, LIM_ULA_Enable :=, LIM_ULA :=, LIM_ULW_Enable :=, LIM_ULW :=, LIM_LLW_Enable :=, LIM_LLW :=, LIM_LLA_Enable :=, LIM_LLA :=, LIM_HYS_Set :=, LIM_HYS :=, INSTANCE := 'CV-51.11', RESTART :=, VISIBILITY :=, OPdwCmd :=, QdwState =>, QOUT =>, QHI_LIM =>, QLO_LIM =>, QLIM_ULA_Enable =>, QLIM_ULA =>, QLIM_ULW_Enable =>, QLIM_ULW =>, QLIM_LLW_Enable =>, QLIM_LLW =>, QLIM_LLA_Enable =>, QLIM_LLA =>, QLIM_HYS =>, QALARM_UL =>, QWARN_UL =>, QWARN_LL =>, QALARM_LL =>, QSIM =>, QLOCK =>, QERR =>, QERR_EXT =>, QERR_OVERRUN =>, QERR_HIGHRANGE =>, QERR_LOWRANGE =>, QERR_WIRE =>, QwAlarm =>)
   END_RUNG
   // the same network as SCL:
   #"CV-51.11"(LIOP_SEL := #Init, L_RESET := #Reset, INSTANCE := 'CV-51.11');   // "Ana_w_K1K2"
END_REGION

REGION Network 15: FT-51.01
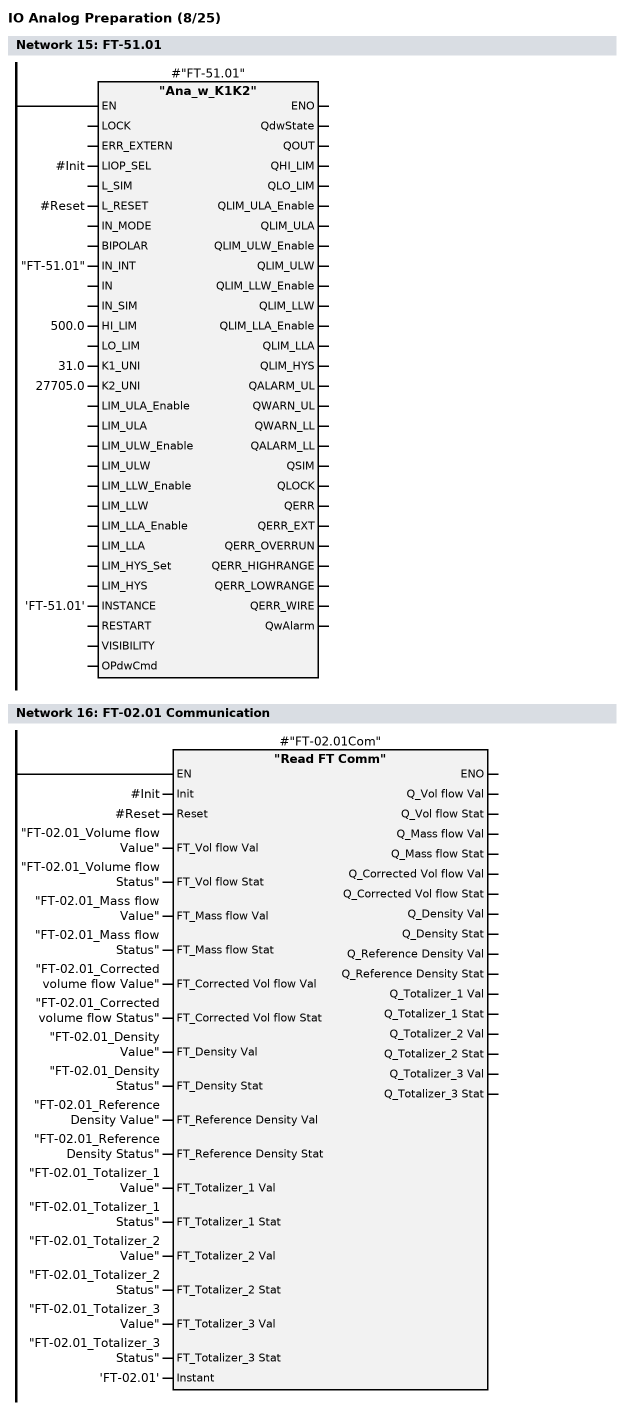
   RUNG wire#powerrail
      #"FT-51.01"(LOCK :=, ERR_EXTERN :=, LIOP_SEL := #Init, L_SIM :=, L_RESET := #Reset, IN_MODE :=, BIPOLAR :=, IN_INT := "FT-51.01", IN :=, IN_SIM :=, HI_LIM := 500.0, LO_LIM :=, K1_UNI := 31.0, K2_UNI := 27705.0, LIM_ULA_Enable :=, LIM_ULA :=, LIM_ULW_Enable :=, LIM_ULW :=, LIM_LLW_Enable :=, LIM_LLW :=, LIM_LLA_Enable :=, LIM_LLA :=, LIM_HYS_Set :=, LIM_HYS :=, INSTANCE := 'FT-51.01', RESTART :=, VISIBILITY :=, OPdwCmd :=, QdwState =>, QOUT =>, QHI_LIM =>, QLO_LIM =>, QLIM_ULA_Enable =>, QLIM_ULA =>, QLIM_ULW_Enable =>, QLIM_ULW =>, QLIM_LLW_Enable =>, QLIM_LLW =>, QLIM_LLA_Enable =>, QLIM_LLA =>, QLIM_HYS =>, QALARM_UL =>, QWARN_UL =>, QWARN_LL =>, QALARM_LL =>, QSIM =>, QLOCK =>, QERR =>, QERR_EXT =>, QERR_OVERRUN =>, QERR_HIGHRANGE =>, QERR_LOWRANGE =>, QERR_WIRE =>, QwAlarm =>)
   END_RUNG
   // the same network as SCL:
   #"FT-51.01"(LIOP_SEL := #Init,   // "Ana_w_K1K2"
               L_RESET := #Reset,
               IN_INT := "FT-51.01",
               HI_LIM := 500.0,
               K1_UNI := 31.0,
               K2_UNI := 27705.0,
               INSTANCE := 'FT-51.01');
END_REGION

REGION Network 16: FT-02.01 Communication
   RUNG wire#powerrail
      #"FT-02.01Com"(Init := #Init, Reset := #Reset, "FT_Vol flow Val" := "FT-02.01_Volume flow Value", "FT_Vol flow Stat" := "FT-02.01_Volume flow Status", "FT_Mass flow Val" := "FT-02.01_Mass flow Value", "FT_Mass flow Stat" := "FT-02.01_Mass flow Status", "FT_Corrected Vol flow Val" := "FT-02.01_Corrected volume flow Value", "FT_Corrected Vol flow Stat" := "FT-02.01_Corrected volume flow Status", "FT_Density Val" := "FT-02.01_Density Value", "FT_Density Stat" := "FT-02.01_Density Status", "FT_Reference Density Val" := "FT-02.01_Reference Density Value", "FT_Reference Density Stat" := "FT-02.01_Reference Density Status", "FT_Totalizer_1 Val" := "FT-02.01_Totalizer_1 Value", "FT_Totalizer_1 Stat" := "FT-02.01_Totalizer_1 Status", "FT_Totalizer_2 Val" := "FT-02.01_Totalizer_2 Value", "FT_Totalizer_2 Stat" := "FT-02.01_Totalizer_2 Status", "FT_Totalizer_3 Val" := "FT-02.01_Totalizer_3 Value", "FT_Totalizer_3 Stat" := "FT-02.01_Totalizer_3 Status", Instant := 'FT-02.01', "Q_Vol flow Val" =>, "Q_Vol flow Stat" =>, "Q_Mass flow Val" =>, "Q_Mass flow Stat" =>, "Q_Corrected Vol flow Val" =>, "Q_Corrected Vol flow Stat" =>, "Q_Density Val" =>, "Q_Density Stat" =>, "Q_Reference Density Val" =>, "Q_Reference Density Stat" =>, "Q_Totalizer_1 Val" =>, "Q_Totalizer_1 Stat" =>, "Q_Totalizer_2 Val" =>, "Q_Totalizer_2 Stat" =>, "Q_Totalizer_3 Val" =>, "Q_Totalizer_3 Stat" =>)
   END_RUNG
   // the same network as SCL:
   #"FT-02.01Com"(Init := #Init,   // "Read FT Comm"
                  Reset := #Reset,
                  "FT_Vol flow Val" := "FT-02.01_Volume flow Value",
                  "FT_Vol flow Stat" := "FT-02.01_Volume flow Status",
                  "FT_Mass flow Val" := "FT-02.01_Mass flow Value",
                  "FT_Mass flow Stat" := "FT-02.01_Mass flow Status",
                  "FT_Corrected Vol flow Val" := "FT-02.01_Corrected volume flow Value",
                  "FT_Corrected Vol flow Stat" := "FT-02.01_Corrected volume flow Status",
                  "FT_Density Val" := "FT-02.01_Density Value",
                  "FT_Density Stat" := "FT-02.01_Density Status",
                  "FT_Reference Density Val" := "FT-02.01_Reference Density Value",
                  "FT_Reference Density Stat" := "FT-02.01_Reference Density Status",
                  "FT_Totalizer_1 Val" := "FT-02.01_Totalizer_1 Value",
                  "FT_Totalizer_1 Stat" := "FT-02.01_Totalizer_1 Status",
                  "FT_Totalizer_2 Val" := "FT-02.01_Totalizer_2 Value",
                  "FT_Totalizer_2 Stat" := "FT-02.01_Totalizer_2 Status",
                  "FT_Totalizer_3 Val" := "FT-02.01_Totalizer_3 Value",
                  "FT_Totalizer_3 Stat" := "FT-02.01_Totalizer_3 Status",
                  Instant := 'FT-02.01');
END_REGION

REGION Network 17: FT-02.01 Flowrate
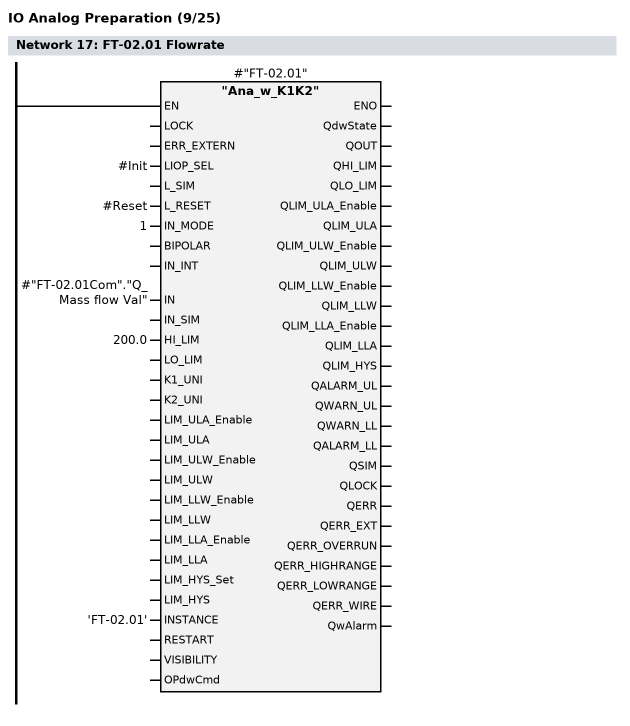
   RUNG wire#powerrail
      #"FT-02.01"(LOCK :=, ERR_EXTERN :=, LIOP_SEL := #Init, L_SIM :=, L_RESET := #Reset, IN_MODE := 1, BIPOLAR :=, IN_INT :=, IN := #"FT-02.01Com"."Q_Mass flow Val", IN_SIM :=, HI_LIM := 200.0, LO_LIM :=, K1_UNI :=, K2_UNI :=, LIM_ULA_Enable :=, LIM_ULA :=, LIM_ULW_Enable :=, LIM_ULW :=, LIM_LLW_Enable :=, LIM_LLW :=, LIM_LLA_Enable :=, LIM_LLA :=, LIM_HYS_Set :=, LIM_HYS :=, INSTANCE := 'FT-02.01', RESTART :=, VISIBILITY :=, OPdwCmd :=, QdwState =>, QOUT =>, QHI_LIM =>, QLO_LIM =>, QLIM_ULA_Enable =>, QLIM_ULA =>, QLIM_ULW_Enable =>, QLIM_ULW =>, QLIM_LLW_Enable =>, QLIM_LLW =>, QLIM_LLA_Enable =>, QLIM_LLA =>, QLIM_HYS =>, QALARM_UL =>, QWARN_UL =>, QWARN_LL =>, QALARM_LL =>, QSIM =>, QLOCK =>, QERR =>, QERR_EXT =>, QERR_OVERRUN =>, QERR_HIGHRANGE =>, QERR_LOWRANGE =>, QERR_WIRE =>, QwAlarm =>)
   END_RUNG
   // the same network as SCL:
   #"FT-02.01"(LIOP_SEL := #Init,   // "Ana_w_K1K2"
               L_RESET := #Reset,
               IN_MODE := 1,
               IN := #"FT-02.01Com"."Q_Mass flow Val",
               HI_LIM := 200.0,
               INSTANCE := 'FT-02.01');
END_REGION

REGION Network 18: FT-03.01 Communication
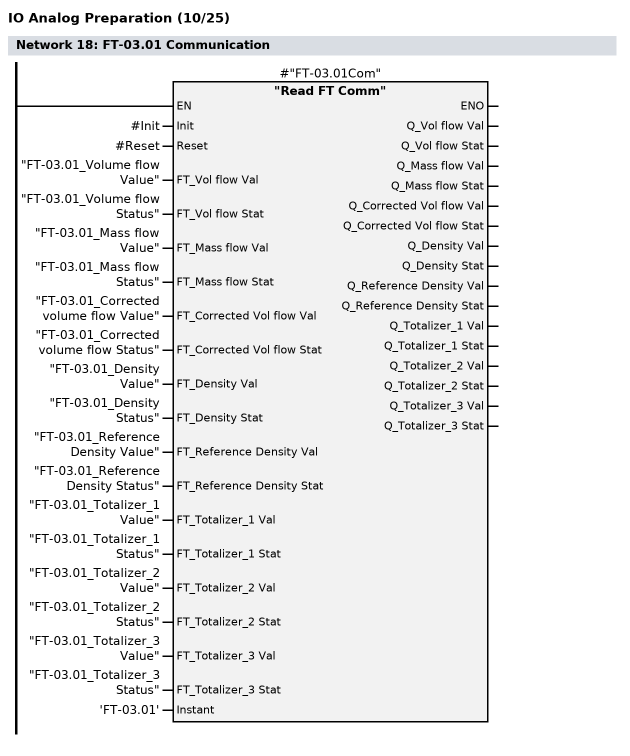
   RUNG wire#powerrail
      #"FT-03.01Com"(Init := #Init, Reset := #Reset, "FT_Vol flow Val" := "FT-03.01_Volume flow Value", "FT_Vol flow Stat" := "FT-03.01_Volume flow Status", "FT_Mass flow Val" := "FT-03.01_Mass flow Value", "FT_Mass flow Stat" := "FT-03.01_Mass flow Status", "FT_Corrected Vol flow Val" := "FT-03.01_Corrected volume flow Value", "FT_Corrected Vol flow Stat" := "FT-03.01_Corrected volume flow Status", "FT_Density Val" := "FT-03.01_Density Value", "FT_Density Stat" := "FT-03.01_Density Status", "FT_Reference Density Val" := "FT-03.01_Reference Density Value", "FT_Reference Density Stat" := "FT-03.01_Reference Density Status", "FT_Totalizer_1 Val" := "FT-03.01_Totalizer_1 Value", "FT_Totalizer_1 Stat" := "FT-03.01_Totalizer_1 Status", "FT_Totalizer_2 Val" := "FT-03.01_Totalizer_2 Value", "FT_Totalizer_2 Stat" := "FT-03.01_Totalizer_2 Status", "FT_Totalizer_3 Val" := "FT-03.01_Totalizer_3 Value", "FT_Totalizer_3 Stat" := "FT-03.01_Totalizer_3 Status", Instant := 'FT-03.01', "Q_Vol flow Val" =>, "Q_Vol flow Stat" =>, "Q_Mass flow Val" =>, "Q_Mass flow Stat" =>, "Q_Corrected Vol flow Val" =>, "Q_Corrected Vol flow Stat" =>, "Q_Density Val" =>, "Q_Density Stat" =>, "Q_Reference Density Val" =>, "Q_Reference Density Stat" =>, "Q_Totalizer_1 Val" =>, "Q_Totalizer_1 Stat" =>, "Q_Totalizer_2 Val" =>, "Q_Totalizer_2 Stat" =>, "Q_Totalizer_3 Val" =>, "Q_Totalizer_3 Stat" =>)
   END_RUNG
   // the same network as SCL:
   #"FT-03.01Com"(Init := #Init,   // "Read FT Comm"
                  Reset := #Reset,
                  "FT_Vol flow Val" := "FT-03.01_Volume flow Value",
                  "FT_Vol flow Stat" := "FT-03.01_Volume flow Status",
                  "FT_Mass flow Val" := "FT-03.01_Mass flow Value",
                  "FT_Mass flow Stat" := "FT-03.01_Mass flow Status",
                  "FT_Corrected Vol flow Val" := "FT-03.01_Corrected volume flow Value",
                  "FT_Corrected Vol flow Stat" := "FT-03.01_Corrected volume flow Status",
                  "FT_Density Val" := "FT-03.01_Density Value",
                  "FT_Density Stat" := "FT-03.01_Density Status",
                  "FT_Reference Density Val" := "FT-03.01_Reference Density Value",
                  "FT_Reference Density Stat" := "FT-03.01_Reference Density Status",
                  "FT_Totalizer_1 Val" := "FT-03.01_Totalizer_1 Value",
                  "FT_Totalizer_1 Stat" := "FT-03.01_Totalizer_1 Status",
                  "FT_Totalizer_2 Val" := "FT-03.01_Totalizer_2 Value",
                  "FT_Totalizer_2 Stat" := "FT-03.01_Totalizer_2 Status",
                  "FT_Totalizer_3 Val" := "FT-03.01_Totalizer_3 Value",
                  "FT_Totalizer_3 Stat" := "FT-03.01_Totalizer_3 Status",
                  Instant := 'FT-03.01');
END_REGION

REGION Network 19: FT-03.01 Flowrate
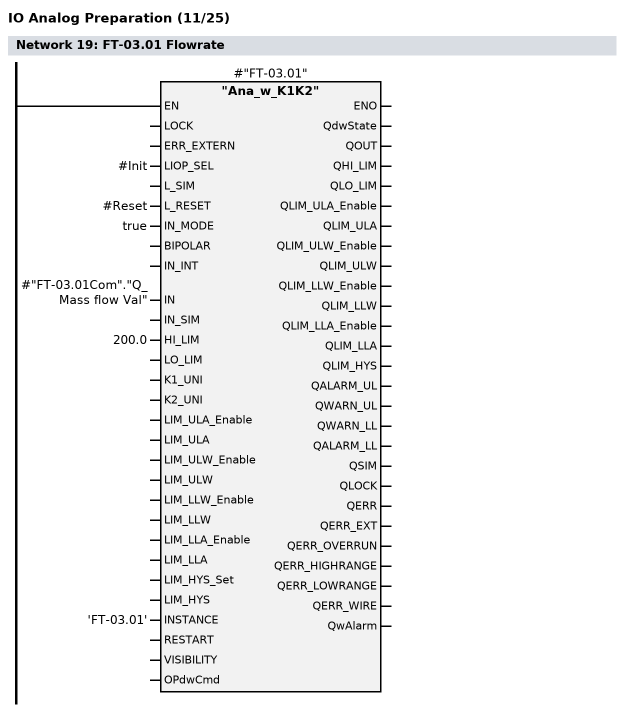
   RUNG wire#powerrail
      #"FT-03.01"(LOCK :=, ERR_EXTERN :=, LIOP_SEL := #Init, L_SIM :=, L_RESET := #Reset, IN_MODE := true, BIPOLAR :=, IN_INT :=, IN := #"FT-03.01Com"."Q_Mass flow Val", IN_SIM :=, HI_LIM := 200.0, LO_LIM :=, K1_UNI :=, K2_UNI :=, LIM_ULA_Enable :=, LIM_ULA :=, LIM_ULW_Enable :=, LIM_ULW :=, LIM_LLW_Enable :=, LIM_LLW :=, LIM_LLA_Enable :=, LIM_LLA :=, LIM_HYS_Set :=, LIM_HYS :=, INSTANCE := 'FT-03.01', RESTART :=, VISIBILITY :=, OPdwCmd :=, QdwState =>, QOUT =>, QHI_LIM =>, QLO_LIM =>, QLIM_ULA_Enable =>, QLIM_ULA =>, QLIM_ULW_Enable =>, QLIM_ULW =>, QLIM_LLW_Enable =>, QLIM_LLW =>, QLIM_LLA_Enable =>, QLIM_LLA =>, QLIM_HYS =>, QALARM_UL =>, QWARN_UL =>, QWARN_LL =>, QALARM_LL =>, QSIM =>, QLOCK =>, QERR =>, QERR_EXT =>, QERR_OVERRUN =>, QERR_HIGHRANGE =>, QERR_LOWRANGE =>, QERR_WIRE =>, QwAlarm =>)
   END_RUNG
   // the same network as SCL:
   #"FT-03.01"(LIOP_SEL := #Init,   // "Ana_w_K1K2"
               L_RESET := #Reset,
               IN_MODE := true,
               IN := #"FT-03.01Com"."Q_Mass flow Val",
               HI_LIM := 200.0,
               INSTANCE := 'FT-03.01');
END_REGION

REGION Network 20: FT-04.01 Communication
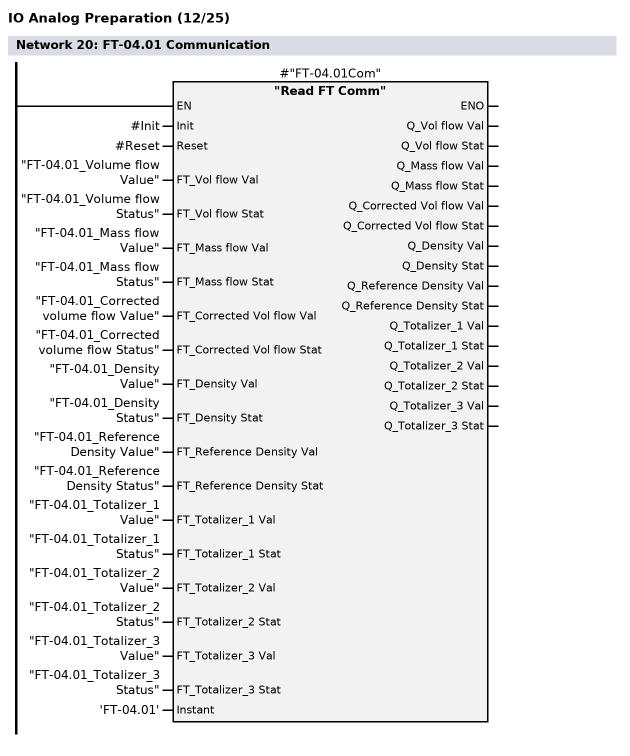
   RUNG wire#powerrail
      #"FT-04.01Com"(Init := #Init, Reset := #Reset, "FT_Vol flow Val" := "FT-04.01_Volume flow Value", "FT_Vol flow Stat" := "FT-04.01_Volume flow Status", "FT_Mass flow Val" := "FT-04.01_Mass flow Value", "FT_Mass flow Stat" := "FT-04.01_Mass flow Status", "FT_Corrected Vol flow Val" := "FT-04.01_Corrected volume flow Value", "FT_Corrected Vol flow Stat" := "FT-04.01_Corrected volume flow Status", "FT_Density Val" := "FT-04.01_Density Value", "FT_Density Stat" := "FT-04.01_Density Status", "FT_Reference Density Val" := "FT-04.01_Reference Density Value", "FT_Reference Density Stat" := "FT-04.01_Reference Density Status", "FT_Totalizer_1 Val" := "FT-04.01_Totalizer_1 Value", "FT_Totalizer_1 Stat" := "FT-04.01_Totalizer_1 Status", "FT_Totalizer_2 Val" := "FT-04.01_Totalizer_2 Value", "FT_Totalizer_2 Stat" := "FT-04.01_Totalizer_2 Status", "FT_Totalizer_3 Val" := "FT-04.01_Totalizer_3 Value", "FT_Totalizer_3 Stat" := "FT-04.01_Totalizer_3 Status", Instant := 'FT-04.01', "Q_Vol flow Val" =>, "Q_Vol flow Stat" =>, "Q_Mass flow Val" =>, "Q_Mass flow Stat" =>, "Q_Corrected Vol flow Val" =>, "Q_Corrected Vol flow Stat" =>, "Q_Density Val" =>, "Q_Density Stat" =>, "Q_Reference Density Val" =>, "Q_Reference Density Stat" =>, "Q_Totalizer_1 Val" =>, "Q_Totalizer_1 Stat" =>, "Q_Totalizer_2 Val" =>, "Q_Totalizer_2 Stat" =>, "Q_Totalizer_3 Val" =>, "Q_Totalizer_3 Stat" =>)
   END_RUNG
   // the same network as SCL:
   #"FT-04.01Com"(Init := #Init,   // "Read FT Comm"
                  Reset := #Reset,
                  "FT_Vol flow Val" := "FT-04.01_Volume flow Value",
                  "FT_Vol flow Stat" := "FT-04.01_Volume flow Status",
                  "FT_Mass flow Val" := "FT-04.01_Mass flow Value",
                  "FT_Mass flow Stat" := "FT-04.01_Mass flow Status",
                  "FT_Corrected Vol flow Val" := "FT-04.01_Corrected volume flow Value",
                  "FT_Corrected Vol flow Stat" := "FT-04.01_Corrected volume flow Status",
                  "FT_Density Val" := "FT-04.01_Density Value",
                  "FT_Density Stat" := "FT-04.01_Density Status",
                  "FT_Reference Density Val" := "FT-04.01_Reference Density Value",
                  "FT_Reference Density Stat" := "FT-04.01_Reference Density Status",
                  "FT_Totalizer_1 Val" := "FT-04.01_Totalizer_1 Value",
                  "FT_Totalizer_1 Stat" := "FT-04.01_Totalizer_1 Status",
                  "FT_Totalizer_2 Val" := "FT-04.01_Totalizer_2 Value",
                  "FT_Totalizer_2 Stat" := "FT-04.01_Totalizer_2 Status",
                  "FT_Totalizer_3 Val" := "FT-04.01_Totalizer_3 Value",
                  "FT_Totalizer_3 Stat" := "FT-04.01_Totalizer_3 Status",
                  Instant := 'FT-04.01');
END_REGION

REGION Network 21: FT-04.01 Flowrate
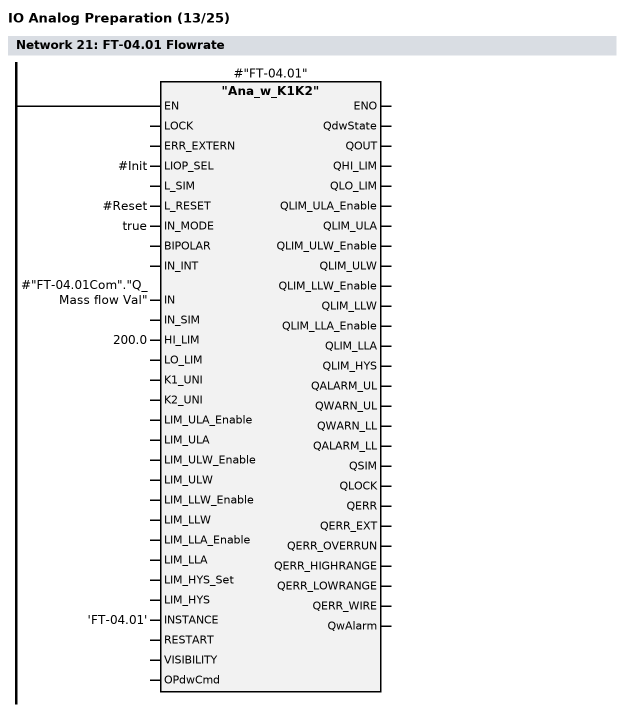
   RUNG wire#powerrail
      #"FT-04.01"(LOCK :=, ERR_EXTERN :=, LIOP_SEL := #Init, L_SIM :=, L_RESET := #Reset, IN_MODE := true, BIPOLAR :=, IN_INT :=, IN := #"FT-04.01Com"."Q_Mass flow Val", IN_SIM :=, HI_LIM := 200.0, LO_LIM :=, K1_UNI :=, K2_UNI :=, LIM_ULA_Enable :=, LIM_ULA :=, LIM_ULW_Enable :=, LIM_ULW :=, LIM_LLW_Enable :=, LIM_LLW :=, LIM_LLA_Enable :=, LIM_LLA :=, LIM_HYS_Set :=, LIM_HYS :=, INSTANCE := 'FT-04.01', RESTART :=, VISIBILITY :=, OPdwCmd :=, QdwState =>, QOUT =>, QHI_LIM =>, QLO_LIM =>, QLIM_ULA_Enable =>, QLIM_ULA =>, QLIM_ULW_Enable =>, QLIM_ULW =>, QLIM_LLW_Enable =>, QLIM_LLW =>, QLIM_LLA_Enable =>, QLIM_LLA =>, QLIM_HYS =>, QALARM_UL =>, QWARN_UL =>, QWARN_LL =>, QALARM_LL =>, QSIM =>, QLOCK =>, QERR =>, QERR_EXT =>, QERR_OVERRUN =>, QERR_HIGHRANGE =>, QERR_LOWRANGE =>, QERR_WIRE =>, QwAlarm =>)
   END_RUNG
   // the same network as SCL:
   #"FT-04.01"(LIOP_SEL := #Init,   // "Ana_w_K1K2"
               L_RESET := #Reset,
               IN_MODE := true,
               IN := #"FT-04.01Com"."Q_Mass flow Val",
               HI_LIM := 200.0,
               INSTANCE := 'FT-04.01');
END_REGION

REGION Network 22: FT-05.01 Communication
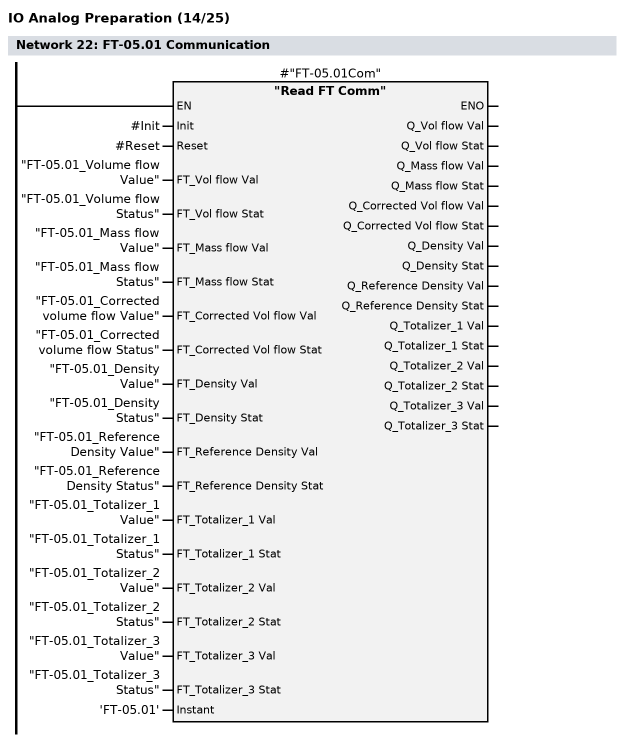
   RUNG wire#powerrail
      #"FT-05.01Com"(Init := #Init, Reset := #Reset, "FT_Vol flow Val" := "FT-05.01_Volume flow Value", "FT_Vol flow Stat" := "FT-05.01_Volume flow Status", "FT_Mass flow Val" := "FT-05.01_Mass flow Value", "FT_Mass flow Stat" := "FT-05.01_Mass flow Status", "FT_Corrected Vol flow Val" := "FT-05.01_Corrected volume flow Value", "FT_Corrected Vol flow Stat" := "FT-05.01_Corrected volume flow Status", "FT_Density Val" := "FT-05.01_Density Value", "FT_Density Stat" := "FT-05.01_Density Status", "FT_Reference Density Val" := "FT-05.01_Reference Density Value", "FT_Reference Density Stat" := "FT-05.01_Reference Density Status", "FT_Totalizer_1 Val" := "FT-05.01_Totalizer_1 Value", "FT_Totalizer_1 Stat" := "FT-05.01_Totalizer_1 Status", "FT_Totalizer_2 Val" := "FT-05.01_Totalizer_2 Value", "FT_Totalizer_2 Stat" := "FT-05.01_Totalizer_2 Status", "FT_Totalizer_3 Val" := "FT-05.01_Totalizer_3 Value", "FT_Totalizer_3 Stat" := "FT-05.01_Totalizer_3 Status", Instant := 'FT-05.01', "Q_Vol flow Val" =>, "Q_Vol flow Stat" =>, "Q_Mass flow Val" =>, "Q_Mass flow Stat" =>, "Q_Corrected Vol flow Val" =>, "Q_Corrected Vol flow Stat" =>, "Q_Density Val" =>, "Q_Density Stat" =>, "Q_Reference Density Val" =>, "Q_Reference Density Stat" =>, "Q_Totalizer_1 Val" =>, "Q_Totalizer_1 Stat" =>, "Q_Totalizer_2 Val" =>, "Q_Totalizer_2 Stat" =>, "Q_Totalizer_3 Val" =>, "Q_Totalizer_3 Stat" =>)
   END_RUNG
   // the same network as SCL:
   #"FT-05.01Com"(Init := #Init,   // "Read FT Comm"
                  Reset := #Reset,
                  "FT_Vol flow Val" := "FT-05.01_Volume flow Value",
                  "FT_Vol flow Stat" := "FT-05.01_Volume flow Status",
                  "FT_Mass flow Val" := "FT-05.01_Mass flow Value",
                  "FT_Mass flow Stat" := "FT-05.01_Mass flow Status",
                  "FT_Corrected Vol flow Val" := "FT-05.01_Corrected volume flow Value",
                  "FT_Corrected Vol flow Stat" := "FT-05.01_Corrected volume flow Status",
                  "FT_Density Val" := "FT-05.01_Density Value",
                  "FT_Density Stat" := "FT-05.01_Density Status",
                  "FT_Reference Density Val" := "FT-05.01_Reference Density Value",
                  "FT_Reference Density Stat" := "FT-05.01_Reference Density Status",
                  "FT_Totalizer_1 Val" := "FT-05.01_Totalizer_1 Value",
                  "FT_Totalizer_1 Stat" := "FT-05.01_Totalizer_1 Status",
                  "FT_Totalizer_2 Val" := "FT-05.01_Totalizer_2 Value",
                  "FT_Totalizer_2 Stat" := "FT-05.01_Totalizer_2 Status",
                  "FT_Totalizer_3 Val" := "FT-05.01_Totalizer_3 Value",
                  "FT_Totalizer_3 Stat" := "FT-05.01_Totalizer_3 Status",
                  Instant := 'FT-05.01');
END_REGION

REGION Network 23: FT-05.01 Flowrate
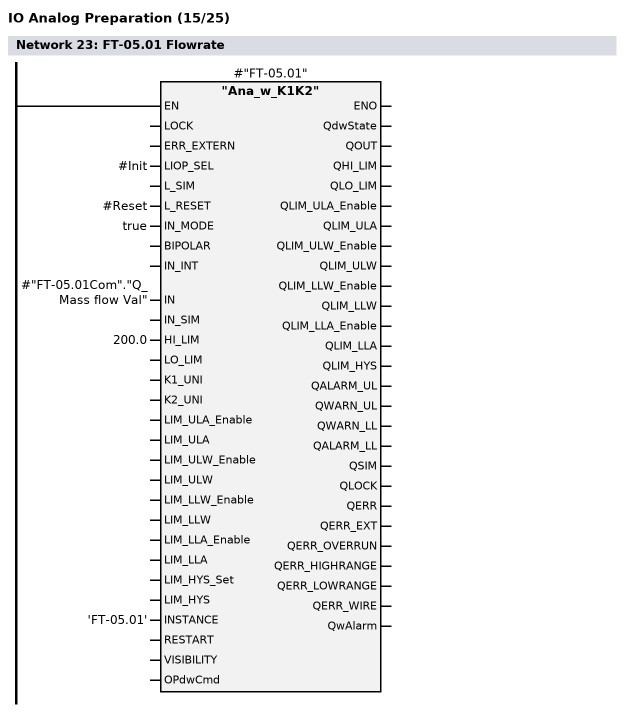
   RUNG wire#powerrail
      #"FT-05.01"(LOCK :=, ERR_EXTERN :=, LIOP_SEL := #Init, L_SIM :=, L_RESET := #Reset, IN_MODE := true, BIPOLAR :=, IN_INT :=, IN := #"FT-05.01Com"."Q_Mass flow Val", IN_SIM :=, HI_LIM := 200.0, LO_LIM :=, K1_UNI :=, K2_UNI :=, LIM_ULA_Enable :=, LIM_ULA :=, LIM_ULW_Enable :=, LIM_ULW :=, LIM_LLW_Enable :=, LIM_LLW :=, LIM_LLA_Enable :=, LIM_LLA :=, LIM_HYS_Set :=, LIM_HYS :=, INSTANCE := 'FT-05.01', RESTART :=, VISIBILITY :=, OPdwCmd :=, QdwState =>, QOUT =>, QHI_LIM =>, QLO_LIM =>, QLIM_ULA_Enable =>, QLIM_ULA =>, QLIM_ULW_Enable =>, QLIM_ULW =>, QLIM_LLW_Enable =>, QLIM_LLW =>, QLIM_LLA_Enable =>, QLIM_LLA =>, QLIM_HYS =>, QALARM_UL =>, QWARN_UL =>, QWARN_LL =>, QALARM_LL =>, QSIM =>, QLOCK =>, QERR =>, QERR_EXT =>, QERR_OVERRUN =>, QERR_HIGHRANGE =>, QERR_LOWRANGE =>, QERR_WIRE =>, QwAlarm =>)
   END_RUNG
   // the same network as SCL:
   #"FT-05.01"(LIOP_SEL := #Init,   // "Ana_w_K1K2"
               L_RESET := #Reset,
               IN_MODE := true,
               IN := #"FT-05.01Com"."Q_Mass flow Val",
               HI_LIM := 200.0,
               INSTANCE := 'FT-05.01');
END_REGION

REGION Network 24: FT-06.01 Communication
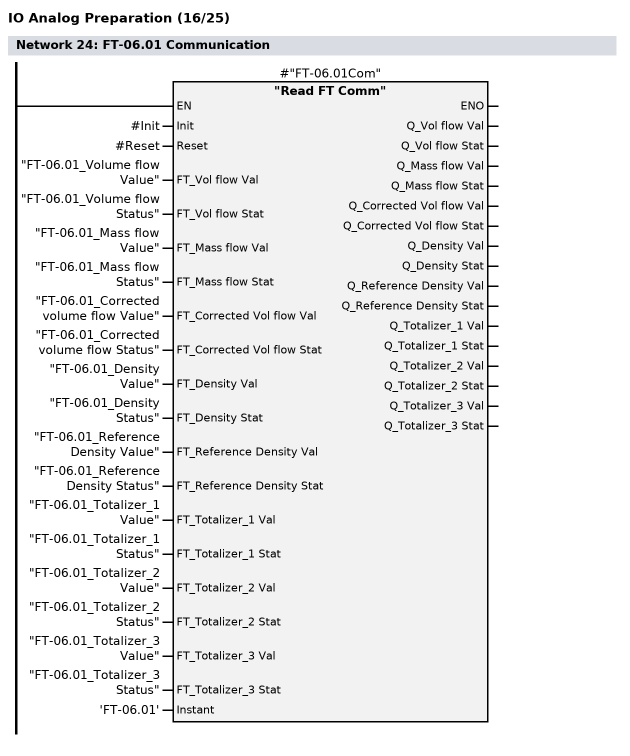
   RUNG wire#powerrail
      #"FT-06.01Com"(Init := #Init, Reset := #Reset, "FT_Vol flow Val" := "FT-06.01_Volume flow Value", "FT_Vol flow Stat" := "FT-06.01_Volume flow Status", "FT_Mass flow Val" := "FT-06.01_Mass flow Value", "FT_Mass flow Stat" := "FT-06.01_Mass flow Status", "FT_Corrected Vol flow Val" := "FT-06.01_Corrected volume flow Value", "FT_Corrected Vol flow Stat" := "FT-06.01_Corrected volume flow Status", "FT_Density Val" := "FT-06.01_Density Value", "FT_Density Stat" := "FT-06.01_Density Status", "FT_Reference Density Val" := "FT-06.01_Reference Density Value", "FT_Reference Density Stat" := "FT-06.01_Reference Density Status", "FT_Totalizer_1 Val" := "FT-06.01_Totalizer_1 Value", "FT_Totalizer_1 Stat" := "FT-06.01_Totalizer_1 Status", "FT_Totalizer_2 Val" := "FT-06.01_Totalizer_2 Value", "FT_Totalizer_2 Stat" := "FT-06.01_Totalizer_2 Status", "FT_Totalizer_3 Val" := "FT-06.01_Totalizer_3 Value", "FT_Totalizer_3 Stat" := "FT-06.01_Totalizer_3 Status", Instant := 'FT-06.01', "Q_Vol flow Val" =>, "Q_Vol flow Stat" =>, "Q_Mass flow Val" =>, "Q_Mass flow Stat" =>, "Q_Corrected Vol flow Val" =>, "Q_Corrected Vol flow Stat" =>, "Q_Density Val" =>, "Q_Density Stat" =>, "Q_Reference Density Val" =>, "Q_Reference Density Stat" =>, "Q_Totalizer_1 Val" =>, "Q_Totalizer_1 Stat" =>, "Q_Totalizer_2 Val" =>, "Q_Totalizer_2 Stat" =>, "Q_Totalizer_3 Val" =>, "Q_Totalizer_3 Stat" =>)
   END_RUNG
   // the same network as SCL:
   #"FT-06.01Com"(Init := #Init,   // "Read FT Comm"
                  Reset := #Reset,
                  "FT_Vol flow Val" := "FT-06.01_Volume flow Value",
                  "FT_Vol flow Stat" := "FT-06.01_Volume flow Status",
                  "FT_Mass flow Val" := "FT-06.01_Mass flow Value",
                  "FT_Mass flow Stat" := "FT-06.01_Mass flow Status",
                  "FT_Corrected Vol flow Val" := "FT-06.01_Corrected volume flow Value",
                  "FT_Corrected Vol flow Stat" := "FT-06.01_Corrected volume flow Status",
                  "FT_Density Val" := "FT-06.01_Density Value",
                  "FT_Density Stat" := "FT-06.01_Density Status",
                  "FT_Reference Density Val" := "FT-06.01_Reference Density Value",
                  "FT_Reference Density Stat" := "FT-06.01_Reference Density Status",
                  "FT_Totalizer_1 Val" := "FT-06.01_Totalizer_1 Value",
                  "FT_Totalizer_1 Stat" := "FT-06.01_Totalizer_1 Status",
                  "FT_Totalizer_2 Val" := "FT-06.01_Totalizer_2 Value",
                  "FT_Totalizer_2 Stat" := "FT-06.01_Totalizer_2 Status",
                  "FT_Totalizer_3 Val" := "FT-06.01_Totalizer_3 Value",
                  "FT_Totalizer_3 Stat" := "FT-06.01_Totalizer_3 Status",
                  Instant := 'FT-06.01');
END_REGION

REGION Network 25: FT-06.01 Flowrate
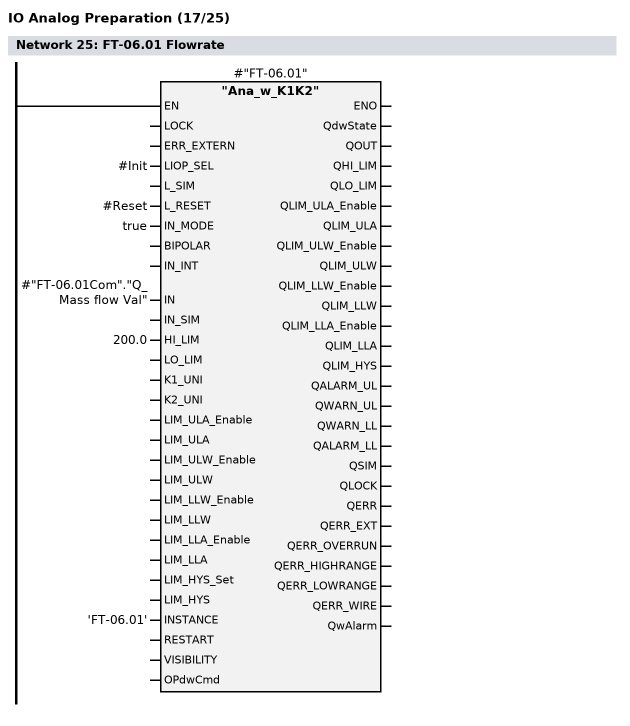
   RUNG wire#powerrail
      #"FT-06.01"(LOCK :=, ERR_EXTERN :=, LIOP_SEL := #Init, L_SIM :=, L_RESET := #Reset, IN_MODE := true, BIPOLAR :=, IN_INT :=, IN := #"FT-06.01Com"."Q_Mass flow Val", IN_SIM :=, HI_LIM := 200.0, LO_LIM :=, K1_UNI :=, K2_UNI :=, LIM_ULA_Enable :=, LIM_ULA :=, LIM_ULW_Enable :=, LIM_ULW :=, LIM_LLW_Enable :=, LIM_LLW :=, LIM_LLA_Enable :=, LIM_LLA :=, LIM_HYS_Set :=, LIM_HYS :=, INSTANCE := 'FT-06.01', RESTART :=, VISIBILITY :=, OPdwCmd :=, QdwState =>, QOUT =>, QHI_LIM =>, QLO_LIM =>, QLIM_ULA_Enable =>, QLIM_ULA =>, QLIM_ULW_Enable =>, QLIM_ULW =>, QLIM_LLW_Enable =>, QLIM_LLW =>, QLIM_LLA_Enable =>, QLIM_LLA =>, QLIM_HYS =>, QALARM_UL =>, QWARN_UL =>, QWARN_LL =>, QALARM_LL =>, QSIM =>, QLOCK =>, QERR =>, QERR_EXT =>, QERR_OVERRUN =>, QERR_HIGHRANGE =>, QERR_LOWRANGE =>, QERR_WIRE =>, QwAlarm =>)
   END_RUNG
   // the same network as SCL:
   #"FT-06.01"(LIOP_SEL := #Init,   // "Ana_w_K1K2"
               L_RESET := #Reset,
               IN_MODE := true,
               IN := #"FT-06.01Com"."Q_Mass flow Val",
               HI_LIM := 200.0,
               INSTANCE := 'FT-06.01');
END_REGION

REGION Network 26: FT-07.01 Communication
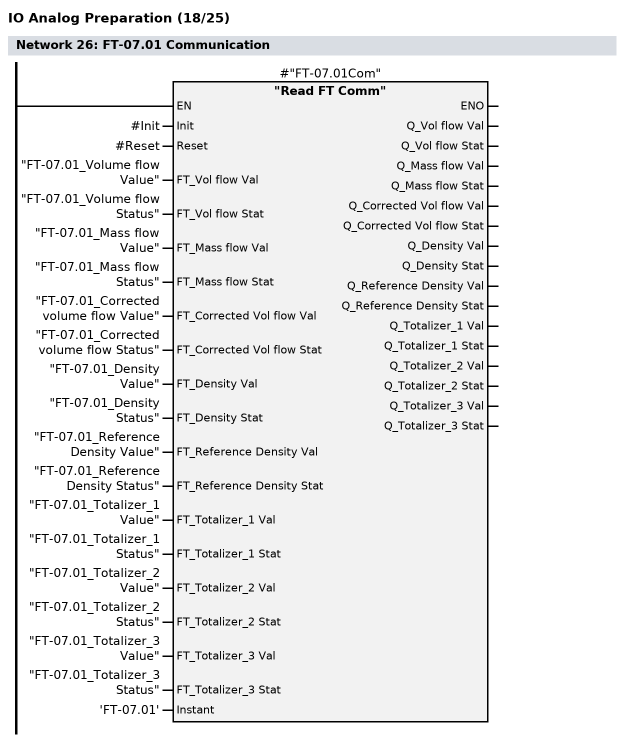
   RUNG wire#powerrail
      #"FT-07.01Com"(Init := #Init, Reset := #Reset, "FT_Vol flow Val" := "FT-07.01_Volume flow Value", "FT_Vol flow Stat" := "FT-07.01_Volume flow Status", "FT_Mass flow Val" := "FT-07.01_Mass flow Value", "FT_Mass flow Stat" := "FT-07.01_Mass flow Status", "FT_Corrected Vol flow Val" := "FT-07.01_Corrected volume flow Value", "FT_Corrected Vol flow Stat" := "FT-07.01_Corrected volume flow Status", "FT_Density Val" := "FT-07.01_Density Value", "FT_Density Stat" := "FT-07.01_Density Status", "FT_Reference Density Val" := "FT-07.01_Reference Density Value", "FT_Reference Density Stat" := "FT-07.01_Reference Density Status", "FT_Totalizer_1 Val" := "FT-07.01_Totalizer_1 Value", "FT_Totalizer_1 Stat" := "FT-07.01_Totalizer_1 Status", "FT_Totalizer_2 Val" := "FT-07.01_Totalizer_2 Value", "FT_Totalizer_2 Stat" := "FT-07.01_Totalizer_2 Status", "FT_Totalizer_3 Val" := "FT-07.01_Totalizer_3 Value", "FT_Totalizer_3 Stat" := "FT-07.01_Totalizer_3 Status", Instant := 'FT-07.01', "Q_Vol flow Val" =>, "Q_Vol flow Stat" =>, "Q_Mass flow Val" =>, "Q_Mass flow Stat" =>, "Q_Corrected Vol flow Val" =>, "Q_Corrected Vol flow Stat" =>, "Q_Density Val" =>, "Q_Density Stat" =>, "Q_Reference Density Val" =>, "Q_Reference Density Stat" =>, "Q_Totalizer_1 Val" =>, "Q_Totalizer_1 Stat" =>, "Q_Totalizer_2 Val" =>, "Q_Totalizer_2 Stat" =>, "Q_Totalizer_3 Val" =>, "Q_Totalizer_3 Stat" =>)
   END_RUNG
   // the same network as SCL:
   #"FT-07.01Com"(Init := #Init,   // "Read FT Comm"
                  Reset := #Reset,
                  "FT_Vol flow Val" := "FT-07.01_Volume flow Value",
                  "FT_Vol flow Stat" := "FT-07.01_Volume flow Status",
                  "FT_Mass flow Val" := "FT-07.01_Mass flow Value",
                  "FT_Mass flow Stat" := "FT-07.01_Mass flow Status",
                  "FT_Corrected Vol flow Val" := "FT-07.01_Corrected volume flow Value",
                  "FT_Corrected Vol flow Stat" := "FT-07.01_Corrected volume flow Status",
                  "FT_Density Val" := "FT-07.01_Density Value",
                  "FT_Density Stat" := "FT-07.01_Density Status",
                  "FT_Reference Density Val" := "FT-07.01_Reference Density Value",
                  "FT_Reference Density Stat" := "FT-07.01_Reference Density Status",
                  "FT_Totalizer_1 Val" := "FT-07.01_Totalizer_1 Value",
                  "FT_Totalizer_1 Stat" := "FT-07.01_Totalizer_1 Status",
                  "FT_Totalizer_2 Val" := "FT-07.01_Totalizer_2 Value",
                  "FT_Totalizer_2 Stat" := "FT-07.01_Totalizer_2 Status",
                  "FT_Totalizer_3 Val" := "FT-07.01_Totalizer_3 Value",
                  "FT_Totalizer_3 Stat" := "FT-07.01_Totalizer_3 Status",
                  Instant := 'FT-07.01');
END_REGION

REGION Network 27: FT-07.01 Flowrate
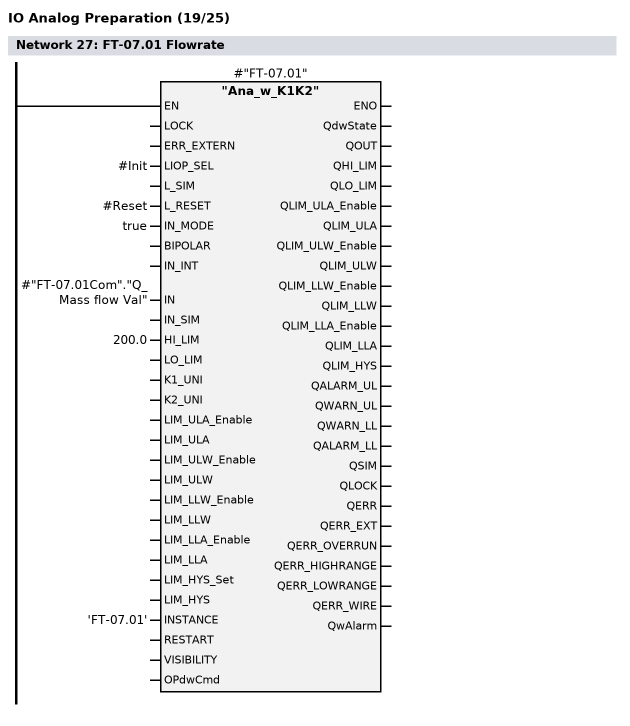
   RUNG wire#powerrail
      #"FT-07.01"(LOCK :=, ERR_EXTERN :=, LIOP_SEL := #Init, L_SIM :=, L_RESET := #Reset, IN_MODE := true, BIPOLAR :=, IN_INT :=, IN := #"FT-07.01Com"."Q_Mass flow Val", IN_SIM :=, HI_LIM := 200.0, LO_LIM :=, K1_UNI :=, K2_UNI :=, LIM_ULA_Enable :=, LIM_ULA :=, LIM_ULW_Enable :=, LIM_ULW :=, LIM_LLW_Enable :=, LIM_LLW :=, LIM_LLA_Enable :=, LIM_LLA :=, LIM_HYS_Set :=, LIM_HYS :=, INSTANCE := 'FT-07.01', RESTART :=, VISIBILITY :=, OPdwCmd :=, QdwState =>, QOUT =>, QHI_LIM =>, QLO_LIM =>, QLIM_ULA_Enable =>, QLIM_ULA =>, QLIM_ULW_Enable =>, QLIM_ULW =>, QLIM_LLW_Enable =>, QLIM_LLW =>, QLIM_LLA_Enable =>, QLIM_LLA =>, QLIM_HYS =>, QALARM_UL =>, QWARN_UL =>, QWARN_LL =>, QALARM_LL =>, QSIM =>, QLOCK =>, QERR =>, QERR_EXT =>, QERR_OVERRUN =>, QERR_HIGHRANGE =>, QERR_LOWRANGE =>, QERR_WIRE =>, QwAlarm =>)
   END_RUNG
   // the same network as SCL:
   #"FT-07.01"(LIOP_SEL := #Init,   // "Ana_w_K1K2"
               L_RESET := #Reset,
               IN_MODE := true,
               IN := #"FT-07.01Com"."Q_Mass flow Val",
               HI_LIM := 200.0,
               INSTANCE := 'FT-07.01');
END_REGION

REGION Network 28: FT-08.01 Communication
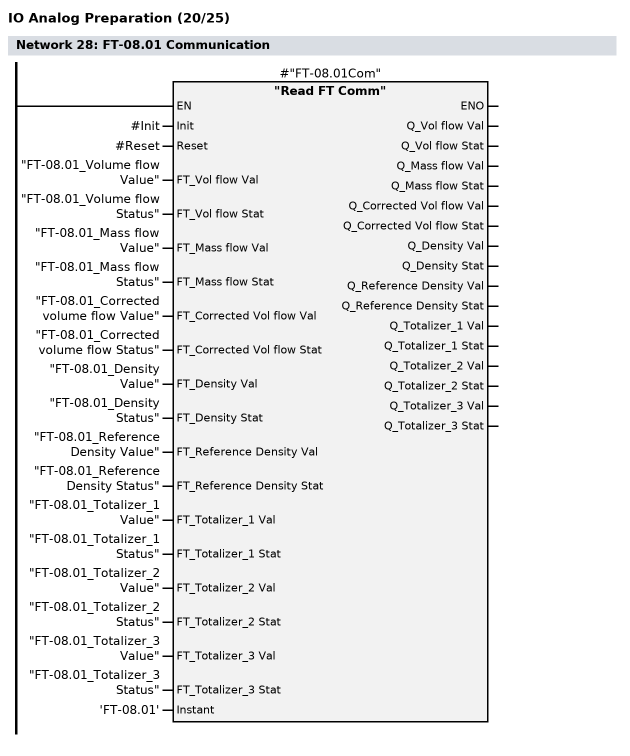
   RUNG wire#powerrail
      #"FT-08.01Com"(Init := #Init, Reset := #Reset, "FT_Vol flow Val" := "FT-08.01_Volume flow Value", "FT_Vol flow Stat" := "FT-08.01_Volume flow Status", "FT_Mass flow Val" := "FT-08.01_Mass flow Value", "FT_Mass flow Stat" := "FT-08.01_Mass flow Status", "FT_Corrected Vol flow Val" := "FT-08.01_Corrected volume flow Value", "FT_Corrected Vol flow Stat" := "FT-08.01_Corrected volume flow Status", "FT_Density Val" := "FT-08.01_Density Value", "FT_Density Stat" := "FT-08.01_Density Status", "FT_Reference Density Val" := "FT-08.01_Reference Density Value", "FT_Reference Density Stat" := "FT-08.01_Reference Density Status", "FT_Totalizer_1 Val" := "FT-08.01_Totalizer_1 Value", "FT_Totalizer_1 Stat" := "FT-08.01_Totalizer_1 Status", "FT_Totalizer_2 Val" := "FT-08.01_Totalizer_2 Value", "FT_Totalizer_2 Stat" := "FT-08.01_Totalizer_2 Status", "FT_Totalizer_3 Val" := "FT-08.01_Totalizer_3 Value", "FT_Totalizer_3 Stat" := "FT-08.01_Totalizer_3 Status", Instant := 'FT-08.01', "Q_Vol flow Val" =>, "Q_Vol flow Stat" =>, "Q_Mass flow Val" =>, "Q_Mass flow Stat" =>, "Q_Corrected Vol flow Val" =>, "Q_Corrected Vol flow Stat" =>, "Q_Density Val" =>, "Q_Density Stat" =>, "Q_Reference Density Val" =>, "Q_Reference Density Stat" =>, "Q_Totalizer_1 Val" =>, "Q_Totalizer_1 Stat" =>, "Q_Totalizer_2 Val" =>, "Q_Totalizer_2 Stat" =>, "Q_Totalizer_3 Val" =>, "Q_Totalizer_3 Stat" =>)
   END_RUNG
   // the same network as SCL:
   #"FT-08.01Com"(Init := #Init,   // "Read FT Comm"
                  Reset := #Reset,
                  "FT_Vol flow Val" := "FT-08.01_Volume flow Value",
                  "FT_Vol flow Stat" := "FT-08.01_Volume flow Status",
                  "FT_Mass flow Val" := "FT-08.01_Mass flow Value",
                  "FT_Mass flow Stat" := "FT-08.01_Mass flow Status",
                  "FT_Corrected Vol flow Val" := "FT-08.01_Corrected volume flow Value",
                  "FT_Corrected Vol flow Stat" := "FT-08.01_Corrected volume flow Status",
                  "FT_Density Val" := "FT-08.01_Density Value",
                  "FT_Density Stat" := "FT-08.01_Density Status",
                  "FT_Reference Density Val" := "FT-08.01_Reference Density Value",
                  "FT_Reference Density Stat" := "FT-08.01_Reference Density Status",
                  "FT_Totalizer_1 Val" := "FT-08.01_Totalizer_1 Value",
                  "FT_Totalizer_1 Stat" := "FT-08.01_Totalizer_1 Status",
                  "FT_Totalizer_2 Val" := "FT-08.01_Totalizer_2 Value",
                  "FT_Totalizer_2 Stat" := "FT-08.01_Totalizer_2 Status",
                  "FT_Totalizer_3 Val" := "FT-08.01_Totalizer_3 Value",
                  "FT_Totalizer_3 Stat" := "FT-08.01_Totalizer_3 Status",
                  Instant := 'FT-08.01');
END_REGION

REGION Network 29: FT-08.01 Flowrate
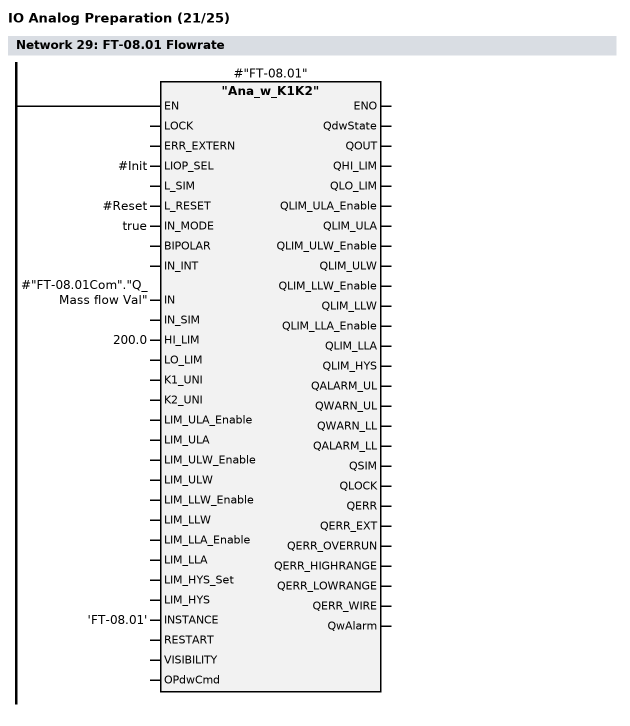
   RUNG wire#powerrail
      #"FT-08.01"(LOCK :=, ERR_EXTERN :=, LIOP_SEL := #Init, L_SIM :=, L_RESET := #Reset, IN_MODE := true, BIPOLAR :=, IN_INT :=, IN := #"FT-08.01Com"."Q_Mass flow Val", IN_SIM :=, HI_LIM := 200.0, LO_LIM :=, K1_UNI :=, K2_UNI :=, LIM_ULA_Enable :=, LIM_ULA :=, LIM_ULW_Enable :=, LIM_ULW :=, LIM_LLW_Enable :=, LIM_LLW :=, LIM_LLA_Enable :=, LIM_LLA :=, LIM_HYS_Set :=, LIM_HYS :=, INSTANCE := 'FT-08.01', RESTART :=, VISIBILITY :=, OPdwCmd :=, QdwState =>, QOUT =>, QHI_LIM =>, QLO_LIM =>, QLIM_ULA_Enable =>, QLIM_ULA =>, QLIM_ULW_Enable =>, QLIM_ULW =>, QLIM_LLW_Enable =>, QLIM_LLW =>, QLIM_LLA_Enable =>, QLIM_LLA =>, QLIM_HYS =>, QALARM_UL =>, QWARN_UL =>, QWARN_LL =>, QALARM_LL =>, QSIM =>, QLOCK =>, QERR =>, QERR_EXT =>, QERR_OVERRUN =>, QERR_HIGHRANGE =>, QERR_LOWRANGE =>, QERR_WIRE =>, QwAlarm =>)
   END_RUNG
   // the same network as SCL:
   #"FT-08.01"(LIOP_SEL := #Init,   // "Ana_w_K1K2"
               L_RESET := #Reset,
               IN_MODE := true,
               IN := #"FT-08.01Com"."Q_Mass flow Val",
               HI_LIM := 200.0,
               INSTANCE := 'FT-08.01');
END_REGION

REGION Network 30: FT-09.01 Communication
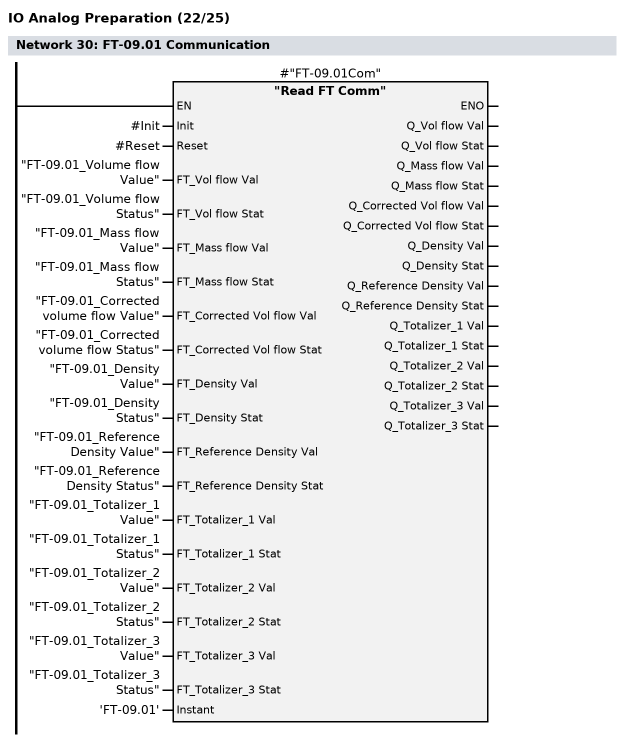
   RUNG wire#powerrail
      #"FT-09.01Com"(Init := #Init, Reset := #Reset, "FT_Vol flow Val" := "FT-09.01_Volume flow Value", "FT_Vol flow Stat" := "FT-09.01_Volume flow Status", "FT_Mass flow Val" := "FT-09.01_Mass flow Value", "FT_Mass flow Stat" := "FT-09.01_Mass flow Status", "FT_Corrected Vol flow Val" := "FT-09.01_Corrected volume flow Value", "FT_Corrected Vol flow Stat" := "FT-09.01_Corrected volume flow Status", "FT_Density Val" := "FT-09.01_Density Value", "FT_Density Stat" := "FT-09.01_Density Status", "FT_Reference Density Val" := "FT-09.01_Reference Density Value", "FT_Reference Density Stat" := "FT-09.01_Reference Density Status", "FT_Totalizer_1 Val" := "FT-09.01_Totalizer_1 Value", "FT_Totalizer_1 Stat" := "FT-09.01_Totalizer_1 Status", "FT_Totalizer_2 Val" := "FT-09.01_Totalizer_2 Value", "FT_Totalizer_2 Stat" := "FT-09.01_Totalizer_2 Status", "FT_Totalizer_3 Val" := "FT-09.01_Totalizer_3 Value", "FT_Totalizer_3 Stat" := "FT-09.01_Totalizer_3 Status", Instant := 'FT-09.01', "Q_Vol flow Val" =>, "Q_Vol flow Stat" =>, "Q_Mass flow Val" =>, "Q_Mass flow Stat" =>, "Q_Corrected Vol flow Val" =>, "Q_Corrected Vol flow Stat" =>, "Q_Density Val" =>, "Q_Density Stat" =>, "Q_Reference Density Val" =>, "Q_Reference Density Stat" =>, "Q_Totalizer_1 Val" =>, "Q_Totalizer_1 Stat" =>, "Q_Totalizer_2 Val" =>, "Q_Totalizer_2 Stat" =>, "Q_Totalizer_3 Val" =>, "Q_Totalizer_3 Stat" =>)
   END_RUNG
   // the same network as SCL:
   #"FT-09.01Com"(Init := #Init,   // "Read FT Comm"
                  Reset := #Reset,
                  "FT_Vol flow Val" := "FT-09.01_Volume flow Value",
                  "FT_Vol flow Stat" := "FT-09.01_Volume flow Status",
                  "FT_Mass flow Val" := "FT-09.01_Mass flow Value",
                  "FT_Mass flow Stat" := "FT-09.01_Mass flow Status",
                  "FT_Corrected Vol flow Val" := "FT-09.01_Corrected volume flow Value",
                  "FT_Corrected Vol flow Stat" := "FT-09.01_Corrected volume flow Status",
                  "FT_Density Val" := "FT-09.01_Density Value",
                  "FT_Density Stat" := "FT-09.01_Density Status",
                  "FT_Reference Density Val" := "FT-09.01_Reference Density Value",
                  "FT_Reference Density Stat" := "FT-09.01_Reference Density Status",
                  "FT_Totalizer_1 Val" := "FT-09.01_Totalizer_1 Value",
                  "FT_Totalizer_1 Stat" := "FT-09.01_Totalizer_1 Status",
                  "FT_Totalizer_2 Val" := "FT-09.01_Totalizer_2 Value",
                  "FT_Totalizer_2 Stat" := "FT-09.01_Totalizer_2 Status",
                  "FT_Totalizer_3 Val" := "FT-09.01_Totalizer_3 Value",
                  "FT_Totalizer_3 Stat" := "FT-09.01_Totalizer_3 Status",
                  Instant := 'FT-09.01');
END_REGION

REGION Network 31: FT-09.01 Flowrate
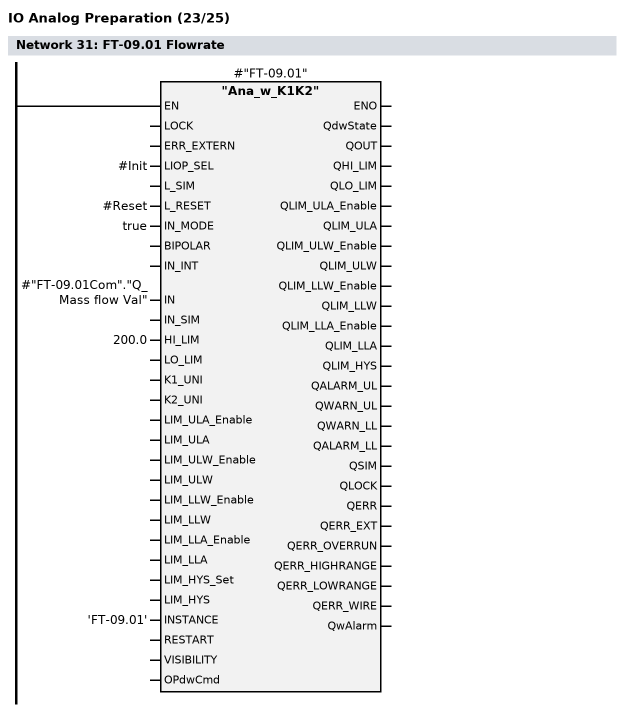
   RUNG wire#powerrail
      #"FT-09.01"(LOCK :=, ERR_EXTERN :=, LIOP_SEL := #Init, L_SIM :=, L_RESET := #Reset, IN_MODE := true, BIPOLAR :=, IN_INT :=, IN := #"FT-09.01Com"."Q_Mass flow Val", IN_SIM :=, HI_LIM := 200.0, LO_LIM :=, K1_UNI :=, K2_UNI :=, LIM_ULA_Enable :=, LIM_ULA :=, LIM_ULW_Enable :=, LIM_ULW :=, LIM_LLW_Enable :=, LIM_LLW :=, LIM_LLA_Enable :=, LIM_LLA :=, LIM_HYS_Set :=, LIM_HYS :=, INSTANCE := 'FT-09.01', RESTART :=, VISIBILITY :=, OPdwCmd :=, QdwState =>, QOUT =>, QHI_LIM =>, QLO_LIM =>, QLIM_ULA_Enable =>, QLIM_ULA =>, QLIM_ULW_Enable =>, QLIM_ULW =>, QLIM_LLW_Enable =>, QLIM_LLW =>, QLIM_LLA_Enable =>, QLIM_LLA =>, QLIM_HYS =>, QALARM_UL =>, QWARN_UL =>, QWARN_LL =>, QALARM_LL =>, QSIM =>, QLOCK =>, QERR =>, QERR_EXT =>, QERR_OVERRUN =>, QERR_HIGHRANGE =>, QERR_LOWRANGE =>, QERR_WIRE =>, QwAlarm =>)
   END_RUNG
   // the same network as SCL:
   #"FT-09.01"(LIOP_SEL := #Init,   // "Ana_w_K1K2"
               L_RESET := #Reset,
               IN_MODE := true,
               IN := #"FT-09.01Com"."Q_Mass flow Val",
               HI_LIM := 200.0,
               INSTANCE := 'FT-09.01');
END_REGION

REGION Network 32: FT-10.01 Communication
